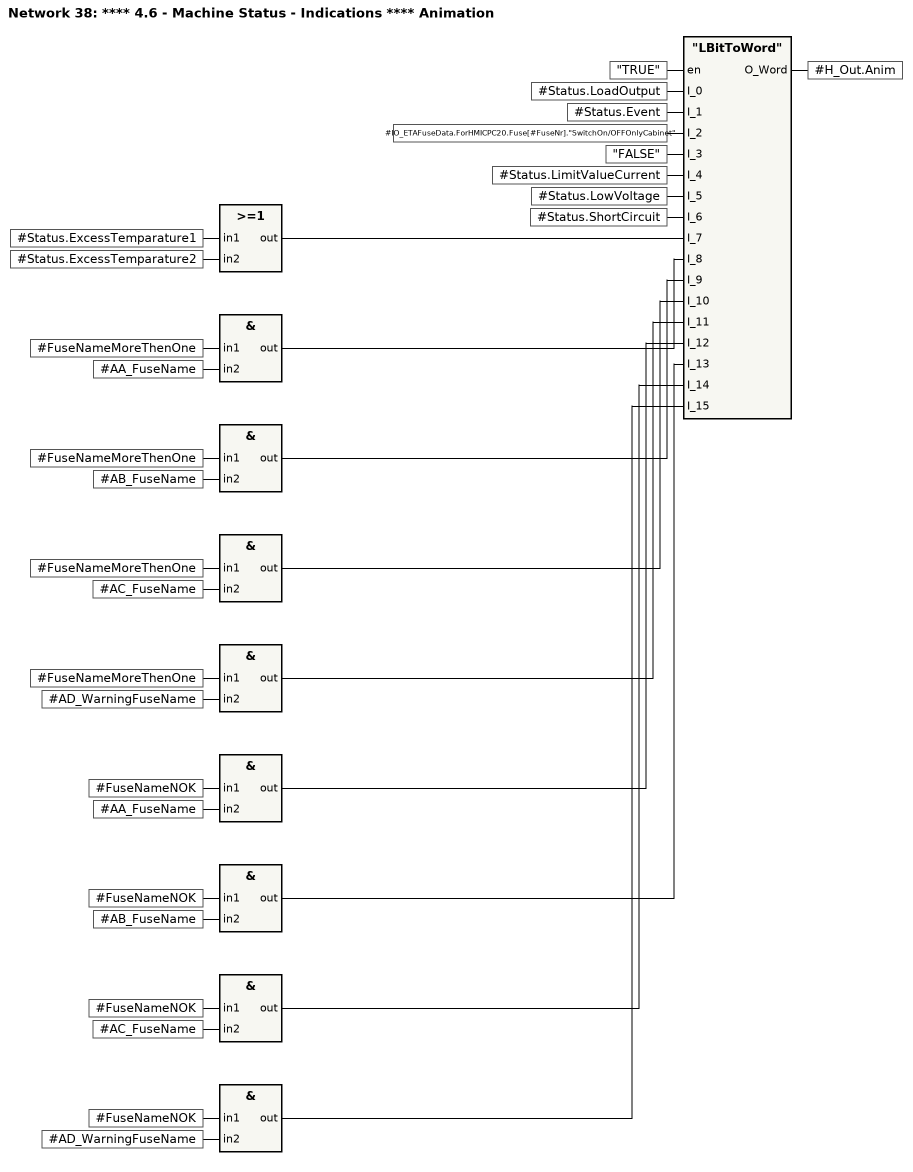
   IF "TRUE" THEN
       "LBitToWord"(I_0 := #Status.LoadOutput,
                    I_1 := #Status.Event,
                    I_2 := #IO_ETAFuseData.ForHMICPC20.Fuse[#FuseNr]."SwitchOn/OFFOnlyCabinet",
                    I_3 := "FALSE",
                    I_4 := #Status.LimitValueCurrent,
                    I_5 := #Status.LowVoltage,
                    I_6 := #Status.ShortCircuit,
                    I_7 := #Status.ExcessTemparature1 OR #Status.ExcessTemparature2,
                    I_8 := #FuseNameMoreThenOne AND #AA_FuseName,
                    I_9 := #FuseNameMoreThenOne AND #AB_FuseName,
                    I_10 := #FuseNameMoreThenOne AND #AC_FuseName,
                    I_11 := #FuseNameMoreThenOne AND #AD_WarningFuseName,
                    I_12 := #FuseNameNOK AND #AA_FuseName,
                    I_13 := #FuseNameNOK AND #AB_FuseName,
                    I_14 := #FuseNameNOK AND #AC_FuseName,
                    I_15 := #FuseNameNOK AND #AD_WarningFuseName,
                    O_Word => #H_Out.Anim);
   END_IF;
END_REGION

REGION Network 39: **** 4.6 - Machine Status - Indications **** Animation2
   // Animation
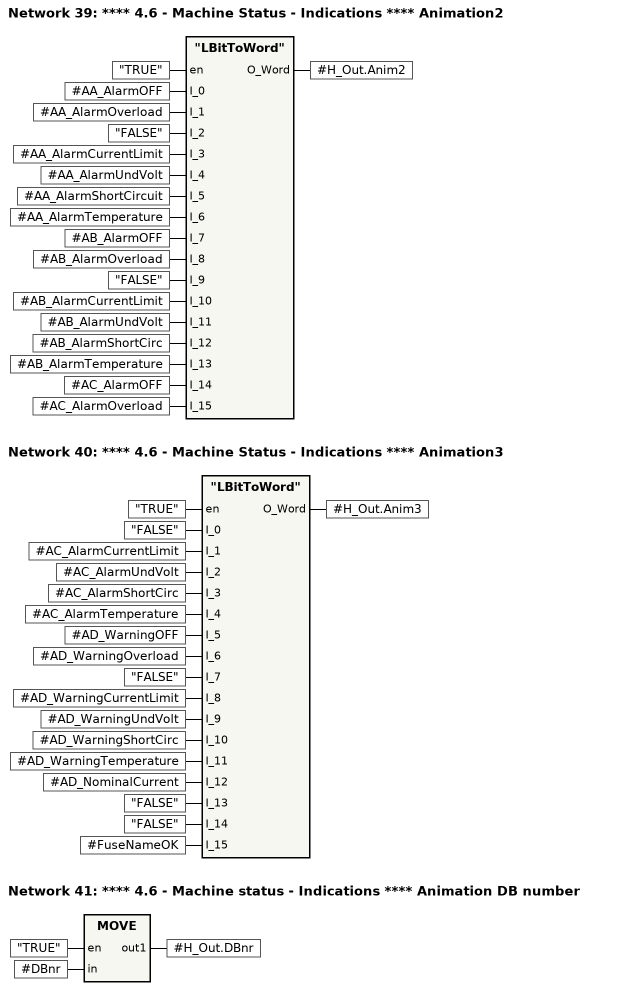
   IF "TRUE" THEN
       "LBitToWord"(I_0 := #AA_AlarmOFF,
                    I_1 := #AA_AlarmOverload,
                    I_2 := "FALSE",
                    I_3 := #AA_AlarmCurrentLimit,
                    I_4 := #AA_AlarmUndVolt,
                    I_5 := #AA_AlarmShortCircuit,
                    I_6 := #AA_AlarmTemperature,
                    I_7 := #AB_AlarmOFF,
                    I_8 := #AB_AlarmOverload,
                    I_9 := "FALSE",
                    I_10 := #AB_AlarmCurrentLimit,
                    I_11 := #AB_AlarmUndVolt,
                    I_12 := #AB_AlarmShortCirc,
                    I_13 := #AB_AlarmTemperature,
                    I_14 := #AC_AlarmOFF,
                    I_15 := #AC_AlarmOverload,
                    O_Word => #H_Out.Anim2);
   END_IF;
END_REGION

REGION Network 40: **** 4.6 - Machine Status - Indications **** Animation3
   // Animation
   IF "TRUE" THEN
       "LBitToWord"(I_0 := "FALSE",
                    I_1 := #AC_AlarmCurrentLimit,
                    I_2 := #AC_AlarmUndVolt,
                    I_3 := #AC_AlarmShortCirc,
                    I_4 := #AC_AlarmTemperature,
                    I_5 := #AD_WarningOFF,
                    I_6 := #AD_WarningOverload,
                    I_7 := "FALSE",
                    I_8 := #AD_WarningCurrentLimit,
                    I_9 := #AD_WarningUndVolt,
                    I_10 := #AD_WarningShortCirc,
                    I_11 := #AD_WarningTemperature,
                    I_12 := #AD_NominalCurrent,
                    I_13 := "FALSE",
                    I_14 := "FALSE",
                    I_15 := #FuseNameOK,
                    O_Word => #H_Out.Anim3);
   END_IF;
END_REGION

REGION Network 41: **** 4.6 - Machine status - Indications **** Animation DB number
   // DB number
   IF "TRUE" THEN #H_Out.DBnr := #DBnr; END_IF;
END_REGION

REGION Network 42: **** 4.6 - Machine Status - Indications **** Animation Fuse Info -> Fuse Number = 0
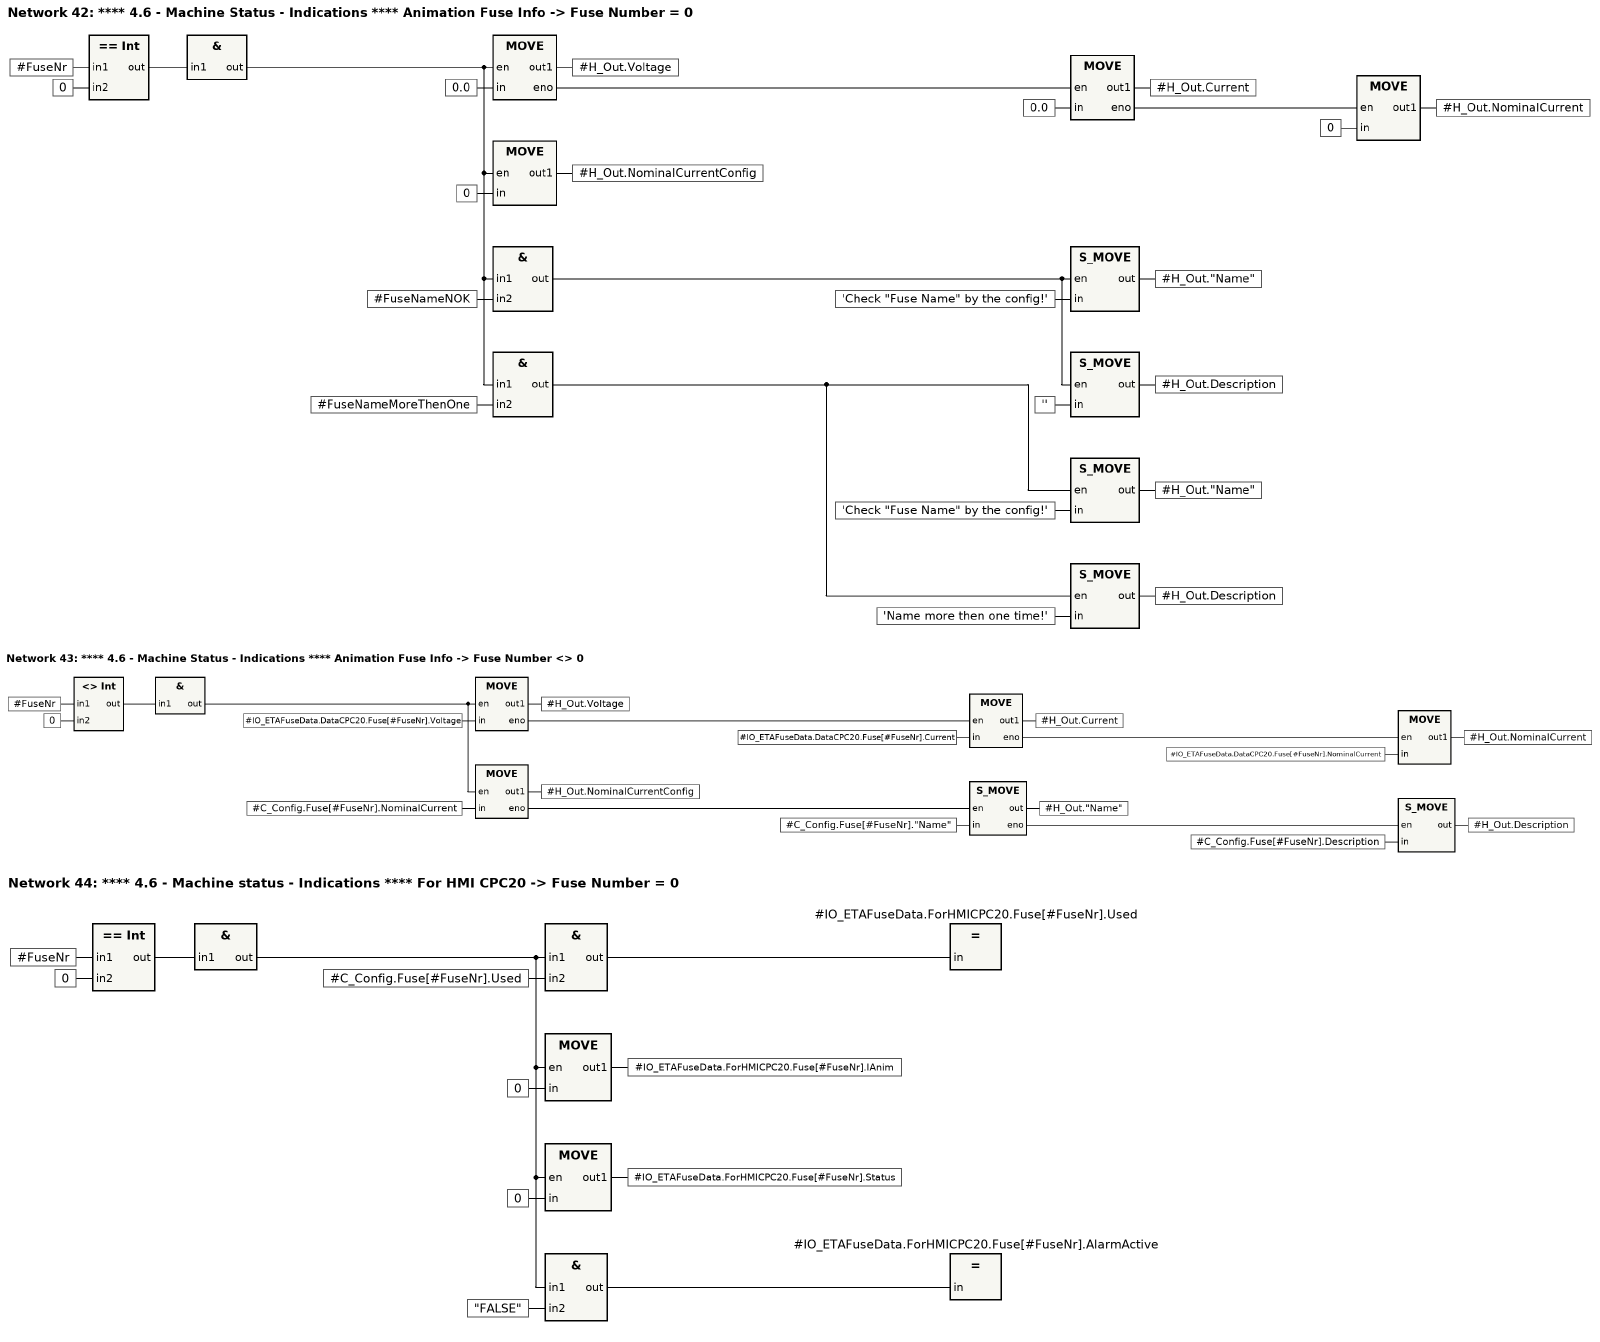
   #_w1 := #FuseNr = 0;
   IF #_w1 THEN
       #H_Out.Voltage := 0.0;
       #H_Out.Current := 0.0;
       #H_Out.NominalCurrent := 0;
       #H_Out.NominalCurrentConfig := 0;
   END_IF;
   IF #_w1 AND #FuseNameNOK THEN
       #H_Out."Name" := 'Check "Fuse Name" by the config!';
       #H_Out.Description := '';
   END_IF;
   IF #_w1 AND #FuseNameMoreThenOne THEN
       #H_Out."Name" := 'Check "Fuse Name" by the config!';
       #H_Out.Description := 'Name more then one time!';
   END_IF;
END_REGION

REGION Network 43: **** 4.6 - Machine Status - Indications **** Animation Fuse Info -> Fuse Number <> 0
   IF #FuseNr <> 0 THEN
       #H_Out.Voltage := #IO_ETAFuseData.DataCPC20.Fuse[#FuseNr].Voltage;
       #H_Out.Current := #IO_ETAFuseData.DataCPC20.Fuse[#FuseNr].Current;
       #H_Out.NominalCurrent := #IO_ETAFuseData.DataCPC20.Fuse[#FuseNr].NominalCurrent;
       #H_Out.NominalCurrentConfig := #C_Config.Fuse[#FuseNr].NominalCurrent;
       #H_Out."Name" := #C_Config.Fuse[#FuseNr]."Name";
       #H_Out.Description := #C_Config.Fuse[#FuseNr].Description;
   END_IF;
END_REGION

REGION Network 44: **** 4.6 - Machine status - Indications **** For HMI CPC20 -> Fuse Number = 0
   #_w1 := #FuseNr = 0;
   #IO_ETAFuseData.ForHMICPC20.Fuse[#FuseNr].Used := #_w1 AND #C_Config.Fuse[#FuseNr].Used;
   IF #_w1 THEN
       #IO_ETAFuseData.ForHMICPC20.Fuse[#FuseNr].IAnim := 0;
       #IO_ETAFuseData.ForHMICPC20.Fuse[#FuseNr].Status := 0;
   END_IF;
   #IO_ETAFuseData.ForHMICPC20.Fuse[#FuseNr].AlarmActive := #_w1 AND "FALSE";
END_REGION

REGION Network 45: **** 4.6 - Machine status - Indications **** For HMI CPC20 -> Fuse Number <> 0
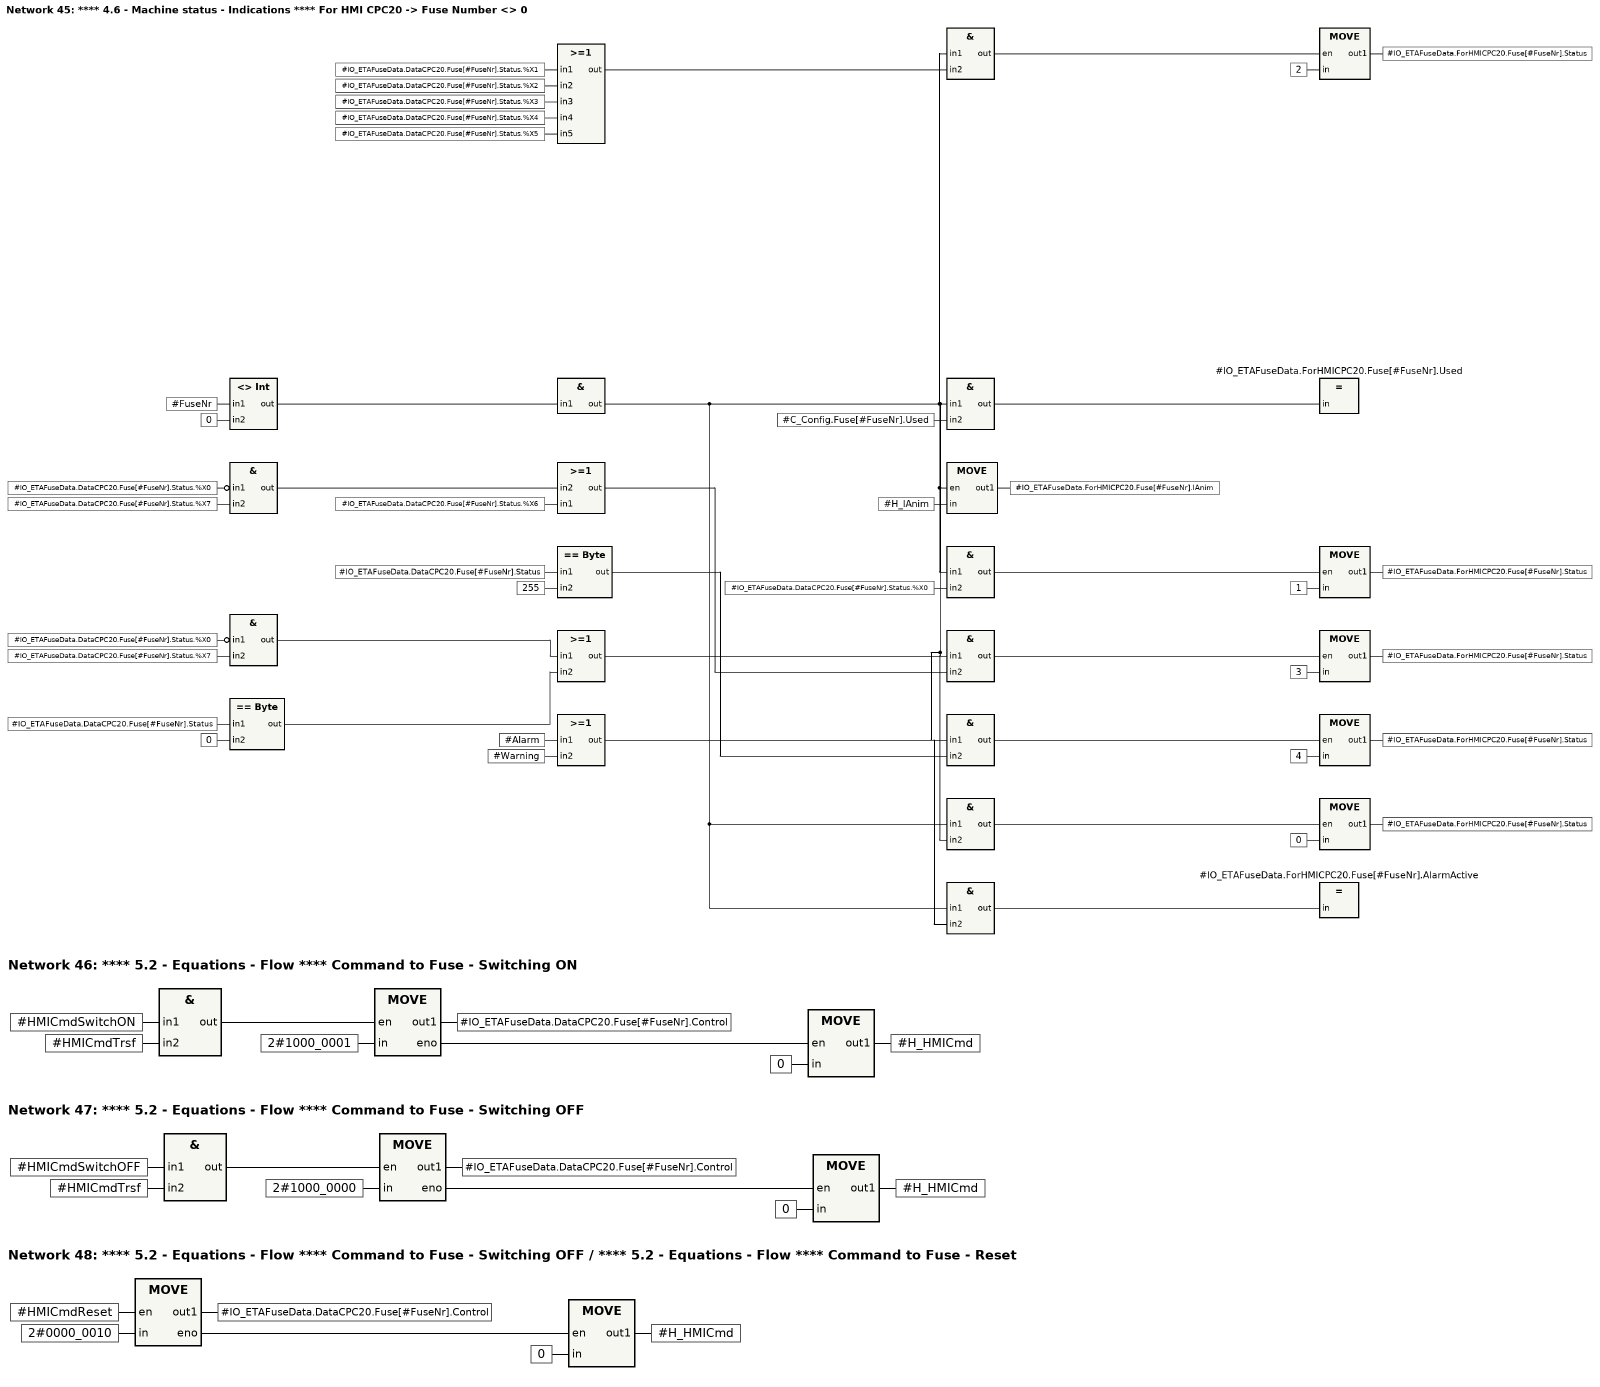
   #_w1 := #FuseNr <> 0;
   #IO_ETAFuseData.ForHMICPC20.Fuse[#FuseNr].Used := #_w1 AND #C_Config.Fuse[#FuseNr].Used;
   IF #_w1 THEN #IO_ETAFuseData.ForHMICPC20.Fuse[#FuseNr].IAnim := #H_IAnim; END_IF;
   IF #_w1 AND #IO_ETAFuseData.DataCPC20.Fuse[#FuseNr].Status.%X0 THEN
       #IO_ETAFuseData.ForHMICPC20.Fuse[#FuseNr].Status := 1;
   END_IF;
   IF #_w1 AND (#IO_ETAFuseData.DataCPC20.Fuse[#FuseNr].Status.%X1 OR #IO_ETAFuseData.DataCPC20.Fuse[#FuseNr].Status.%X2 OR #IO_ETAFuseData.DataCPC20.Fuse[#FuseNr].Status.%X3 OR #IO_ETAFuseData.DataCPC20.Fuse[#FuseNr].Status.%X4 OR #IO_ETAFuseData.DataCPC20.Fuse[#FuseNr].Status.%X5) THEN
       #IO_ETAFuseData.ForHMICPC20.Fuse[#FuseNr].Status := 2;
   END_IF;
   IF #_w1 AND ((NOT #IO_ETAFuseData.DataCPC20.Fuse[#FuseNr].Status.%X0 AND #IO_ETAFuseData.DataCPC20.Fuse[#FuseNr].Status.%X7) OR #IO_ETAFuseData.DataCPC20.Fuse[#FuseNr].Status.%X6) THEN
       #IO_ETAFuseData.ForHMICPC20.Fuse[#FuseNr].Status := 3;
   END_IF;
   IF #_w1 AND (#IO_ETAFuseData.DataCPC20.Fuse[#FuseNr].Status = 255) THEN
       #IO_ETAFuseData.ForHMICPC20.Fuse[#FuseNr].Status := 4;
   END_IF;
   IF #_w1 AND ((NOT #IO_ETAFuseData.DataCPC20.Fuse[#FuseNr].Status.%X0 AND #IO_ETAFuseData.DataCPC20.Fuse[#FuseNr].Status.%X7) OR (#IO_ETAFuseData.DataCPC20.Fuse[#FuseNr].Status = 0)) THEN
       #IO_ETAFuseData.ForHMICPC20.Fuse[#FuseNr].Status := 0;
   END_IF;
   #IO_ETAFuseData.ForHMICPC20.Fuse[#FuseNr].AlarmActive := #_w1 AND (#Alarm OR #Warning);
END_REGION

REGION Network 46: **** 5.2 - Equations - Flow **** Command to Fuse - Switching ON
   // Switching ON
   // ENO of a box is taken as its EN; it also drops when the box reports an error
   IF #HMICmdSwitchON AND #HMICmdTrsf THEN
       #IO_ETAFuseData.DataCPC20.Fuse[#FuseNr].Control := 2#1000_0001;
       #H_HMICmd := 0;
   END_IF;
END_REGION

REGION Network 47: **** 5.2 - Equations - Flow **** Command to Fuse - Switching OFF
   // Switching OFF
   // ENO of a box is taken as its EN; it also drops when the box reports an error
   IF #HMICmdSwitchOFF AND #HMICmdTrsf THEN
       #IO_ETAFuseData.DataCPC20.Fuse[#FuseNr].Control := 2#1000_0000;
       #H_HMICmd := 0;
   END_IF;
END_REGION

REGION Network 48: **** 5.2 - Equations - Flow **** Command to Fuse - Switching OFF / **** 5.2 - Equations - Flow **** Command to Fuse - Reset
   // Switching OFF / Reset
   // ENO of a box is taken as its EN; it also drops when the box reports an error
   IF #HMICmdReset THEN
       #IO_ETAFuseData.DataCPC20.Fuse[#FuseNr].Control := 2#0000_0010;
       #H_HMICmd := 0;
   END_IF;
END_REGION

REGION Network 49: **** 5.2 - Equations - Flow **** Command to Fuse - Reset Control
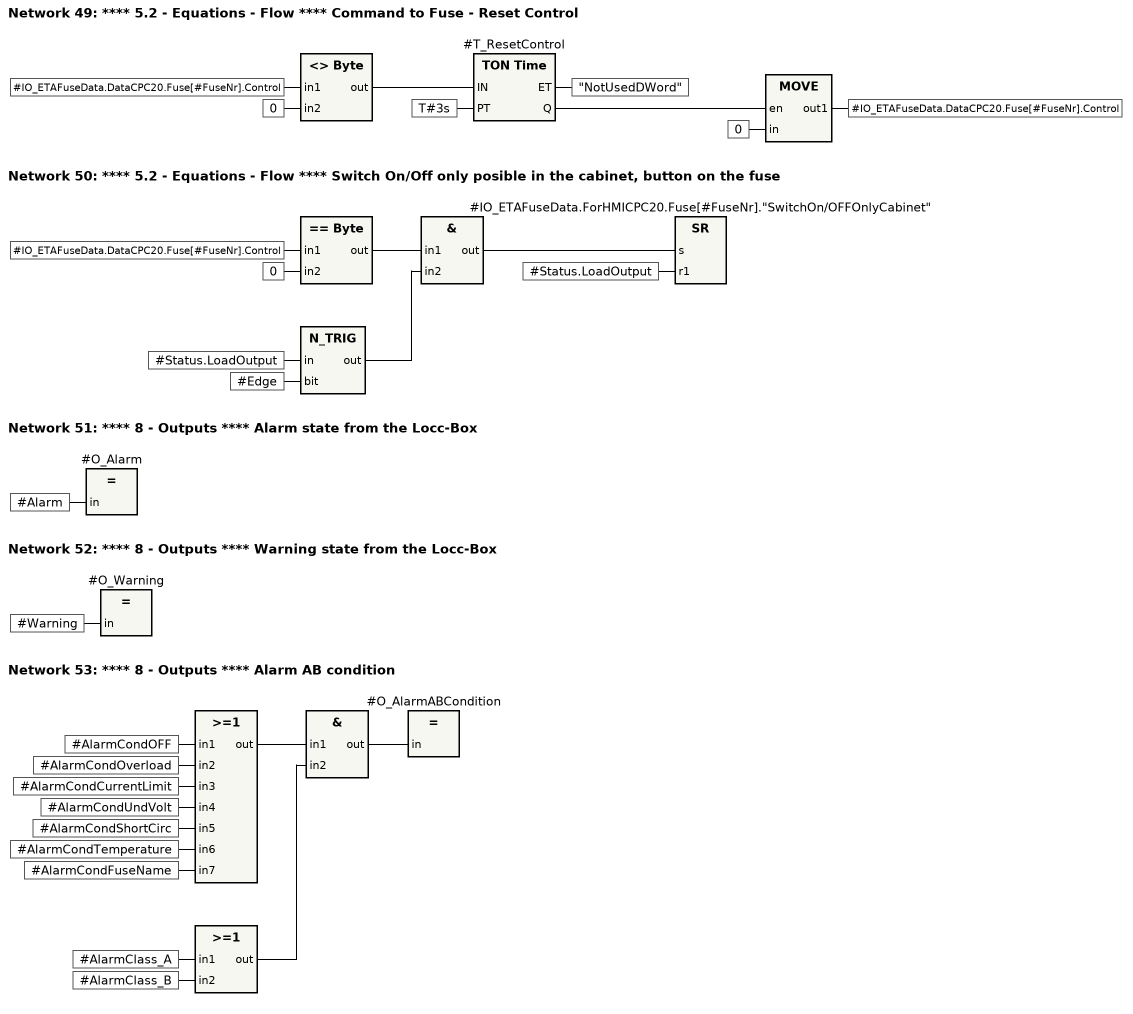
   #T_ResetControl(IN := #IO_ETAFuseData.DataCPC20.Fuse[#FuseNr].Control <> 0, PT := T#3s, ET => "NotUsedDWord");   // TON
   IF #T_ResetControl.Q THEN #IO_ETAFuseData.DataCPC20.Fuse[#FuseNr].Control := 0; END_IF;
END_REGION

REGION Network 50: **** 5.2 - Equations - Flow **** Switch On/Off only posible in the cabinet, button on the fuse
   #_w1 := NOT #Status.LoadOutput AND #Edge;   // falling edge
   #Edge := #Status.LoadOutput;
   IF (#IO_ETAFuseData.DataCPC20.Fuse[#FuseNr].Control = 0) AND #_w1 THEN
       #IO_ETAFuseData.ForHMICPC20.Fuse[#FuseNr]."SwitchOn/OFFOnlyCabinet" := TRUE;   // SR flip-flop
   END_IF;
   IF #Status.LoadOutput THEN
       #IO_ETAFuseData.ForHMICPC20.Fuse[#FuseNr]."SwitchOn/OFFOnlyCabinet" := FALSE;
   END_IF;
END_REGION

REGION Network 51: **** 8 - Outputs **** Alarm state from the Locc-Box
   // Alarm state from the Locc-Box
   #O_Alarm := #Alarm;
END_REGION

REGION Network 52: **** 8 - Outputs **** Warning state from the Locc-Box
   // Warning state from the Locc-Box
   #O_Warning := #Warning;
END_REGION

REGION Network 53: **** 8 - Outputs **** Alarm AB condition
   // Alarm AB condition
   #O_AlarmABCondition := (#AlarmCondOFF OR #AlarmCondOverload OR #AlarmCondCurrentLimit OR #AlarmCondUndVolt OR #AlarmCondShortCirc OR #AlarmCondTemperature OR #AlarmCondFuseName) AND (#AlarmClass_A OR #AlarmClass_B);
END_REGION

REGION Network 54: **** 9.2 - Alarm DWord**** Alarm To DWord
   // Alarm Word
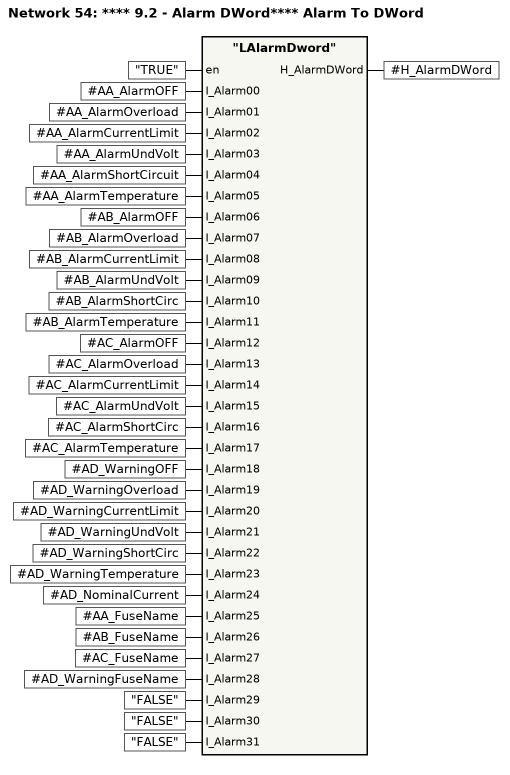
   IF "TRUE" THEN
       "LAlarmDword"(I_Alarm00 := #AA_AlarmOFF,
                     I_Alarm01 := #AA_AlarmOverload,
                     I_Alarm02 := #AA_AlarmCurrentLimit,
                     I_Alarm03 := #AA_AlarmUndVolt,
                     I_Alarm04 := #AA_AlarmShortCircuit,
                     I_Alarm05 := #AA_AlarmTemperature,
                     I_Alarm06 := #AB_AlarmOFF,
                     I_Alarm07 := #AB_AlarmOverload,
                     I_Alarm08 := #AB_AlarmCurrentLimit,
                     I_Alarm09 := #AB_AlarmUndVolt,
                     I_Alarm10 := #AB_AlarmShortCirc,
                     I_Alarm11 := #AB_AlarmTemperature,
                     I_Alarm12 := #AC_AlarmOFF,
                     I_Alarm13 := #AC_AlarmOverload,
                     I_Alarm14 := #AC_AlarmCurrentLimit,
                     I_Alarm15 := #AC_AlarmUndVolt,
                     I_Alarm16 := #AC_AlarmShortCirc,
                     I_Alarm17 := #AC_AlarmTemperature,
                     I_Alarm18 := #AD_WarningOFF,
                     I_Alarm19 := #AD_WarningOverload,
                     I_Alarm20 := #AD_WarningCurrentLimit,
                     I_Alarm21 := #AD_WarningUndVolt,
                     I_Alarm22 := #AD_WarningShortCirc,
                     I_Alarm23 := #AD_WarningTemperature,
                     I_Alarm24 := #AD_NominalCurrent,
                     I_Alarm25 := #AA_FuseName,
                     I_Alarm26 := #AB_FuseName,
                     I_Alarm27 := #AC_FuseName,
                     I_Alarm28 := #AD_WarningFuseName,
                     I_Alarm29 := "FALSE",
                     I_Alarm30 := "FALSE",
                     I_Alarm31 := "FALSE",
                     H_AlarmDWord => #H_AlarmDWord);
   END_IF;
END_REGION
END_FUNCTION_BLOCK

FUNCTION_BLOCK "LGapControlAlarm"   // FB1415, FBD
TITLE = LGapControlAlarm
{ S7_Optimized_Access := 'FALSE' }
AUTHOR : VCC
FAMILY : AlarmHnd
NAME : GapCtrl
VERSION : 1.0
// ================================================================================
// This module is used everywhere one alarm shall be generated when one input 
// photocell becomes false and this photocell signal has to be checked during 
// transfer.
// If the alarm is enable, the photocell may not be deactivated by means of 
// breaking the ray.
// This FB also check the consistency of the photocell. During the period we are 
// sure the photocell must be activated (transfer), the input of the photocell is 
// checked on activity.
// Alarm is disable from HMI, a boolean output is available to inform the upper 
// level and do action in the Alarm summary.
// When the conditions to generate the alarm is disappear, a boolean output is 
// available to inform the upper level that the alarm can be reset.
// The alarm is reset by means of the AlarmResetPB signal.
// ================================================================================
// stored: AutoNumber false, IsIECCheckEnabled false, SetENOAutomatically False, UDAEnableTagReadback false
   VAR_INPUT
      I_GapControl { ExternalAccessible := 'False'; ExternalVisible := 'False'; ExternalWritable := 'False'} : Bool;   // Input signal of the alarm
      I_CheckGapCtrlTrueCond { ExternalAccessible := 'False'; ExternalVisible := 'False'; ExternalWritable := 'False'} : Bool;   // Condition to check gap control photocell on TRUE
      I_CheckGapCtrlFalseCond { ExternalAccessible := 'False'; ExternalVisible := 'False'; ExternalWritable := 'False'} : Bool;   // Condition ot check gap control photocell on FALSE
      I_EnableAlarm { ExternalAccessible := 'False'; ExternalVisible := 'False'; ExternalWritable := 'False'} : Bool := TRUE;   // Enable alarm from upper level
      I_Invisible { ExternalAccessible := 'False'; ExternalVisible := 'False'; ExternalWritable := 'False'} : Bool;   // Invisible
      I_AlarmResetPB { ExternalAccessible := 'False'; ExternalVisible := 'False'; ExternalWritable := 'False'} : Bool;   // Alarm reset pushbutton is activated
   END_VAR
   VAR_OUTPUT
      O_GapControlAlm { ExternalAccessible := 'False'; ExternalVisible := 'False'; ExternalWritable := 'False'} : Bool;   // Gap control Alarm
      O_GapControlTrueAlm { ExternalAccessible := 'False'; ExternalVisible := 'False'; ExternalWritable := 'False'} : Bool;   // Gap control True Alarm
      O_GapControlFalseAlm { ExternalAccessible := 'False'; ExternalVisible := 'False'; ExternalWritable := 'False'} : Bool;   // Gap control False Alarm
      O_AlarmDisabled { ExternalAccessible := 'False'; ExternalVisible := 'False'; ExternalWritable := 'False'} : Bool;   // Alarm disabled from HMI
      O_AlarmABCondition { ExternalAccessible := 'False'; ExternalVisible := 'False'; ExternalWritable := 'False'} : Bool;   // Alarm AB condition
      H_IAnim { ExternalAccessible := 'False'; ExternalVisible := 'False'; ExternalWritable := 'False'} : Word;
   END_VAR
   VAR DB_SPECIFIC
      H_In : Struct   // HMI
         DisableAlarm : Bool;   // Disable alarm from HMI
      END_STRUCT;
      H_Out : Struct   // HMI
         Anim : Word;   // HMI Animation of the object
      END_STRUCT;
      GapControlAlm { ExternalAccessible := 'False'; ExternalVisible := 'False'; ExternalWritable := 'False'} : Bool;   // Gap control Alarm
      GapControlAlmCond { ExternalAccessible := 'False'; ExternalVisible := 'False'; ExternalWritable := 'False'} : Bool;   // Gap control Alarm condition
      PCheckGapTrue { ExternalAccessible := 'False'; ExternalVisible := 'False'; ExternalWritable := 'False'} : Bool;   // Pulse Check detection on True signal
      GapControlTrueMem { ExternalAccessible := 'False'; ExternalVisible := 'False'; ExternalWritable := 'False'} : Bool;   // Memory Gap control on True signal
      GapControlTrueAlm { ExternalAccessible := 'False'; ExternalVisible := 'False'; ExternalWritable := 'False'} : Bool;   // Gap control alarm on True
      GapControlTrueAlmCond { ExternalAccessible := 'False'; ExternalVisible := 'False'; ExternalWritable := 'False'} : Bool;   // Alarm condition of Gap Control True Alarm
      PCheckGapfalse { ExternalAccessible := 'False'; ExternalVisible := 'False'; ExternalWritable := 'False'} : Bool;   // Pulse Check detection on False signal
      GapControlFalseMem { ExternalAccessible := 'False'; ExternalVisible := 'False'; ExternalWritable := 'False'} : Bool;   // Memory Gap control on False signal
      GapControlFalseAlm { ExternalAccessible := 'False'; ExternalVisible := 'False'; ExternalWritable := 'False'} : Bool;   // Gap control alarm on False
      GapControlFalseAlmCond { ExternalAccessible := 'False'; ExternalVisible := 'False'; ExternalWritable := 'False'} : Bool;   // Alarm condition of Gap Control False Alarm
   END_VAR
   VAR_TEMP   // added for the SCL form of the ladder/FBD networks
      _w1 : Bool;
   END_VAR
BEGIN

REGION Network 1: **** 2.2 - Alarms - Alarms Generation **** Condition of the Gap control alarm for the Normal CLOSED input
   // Condition of the Gap control alarm for the Normal CLOSED input
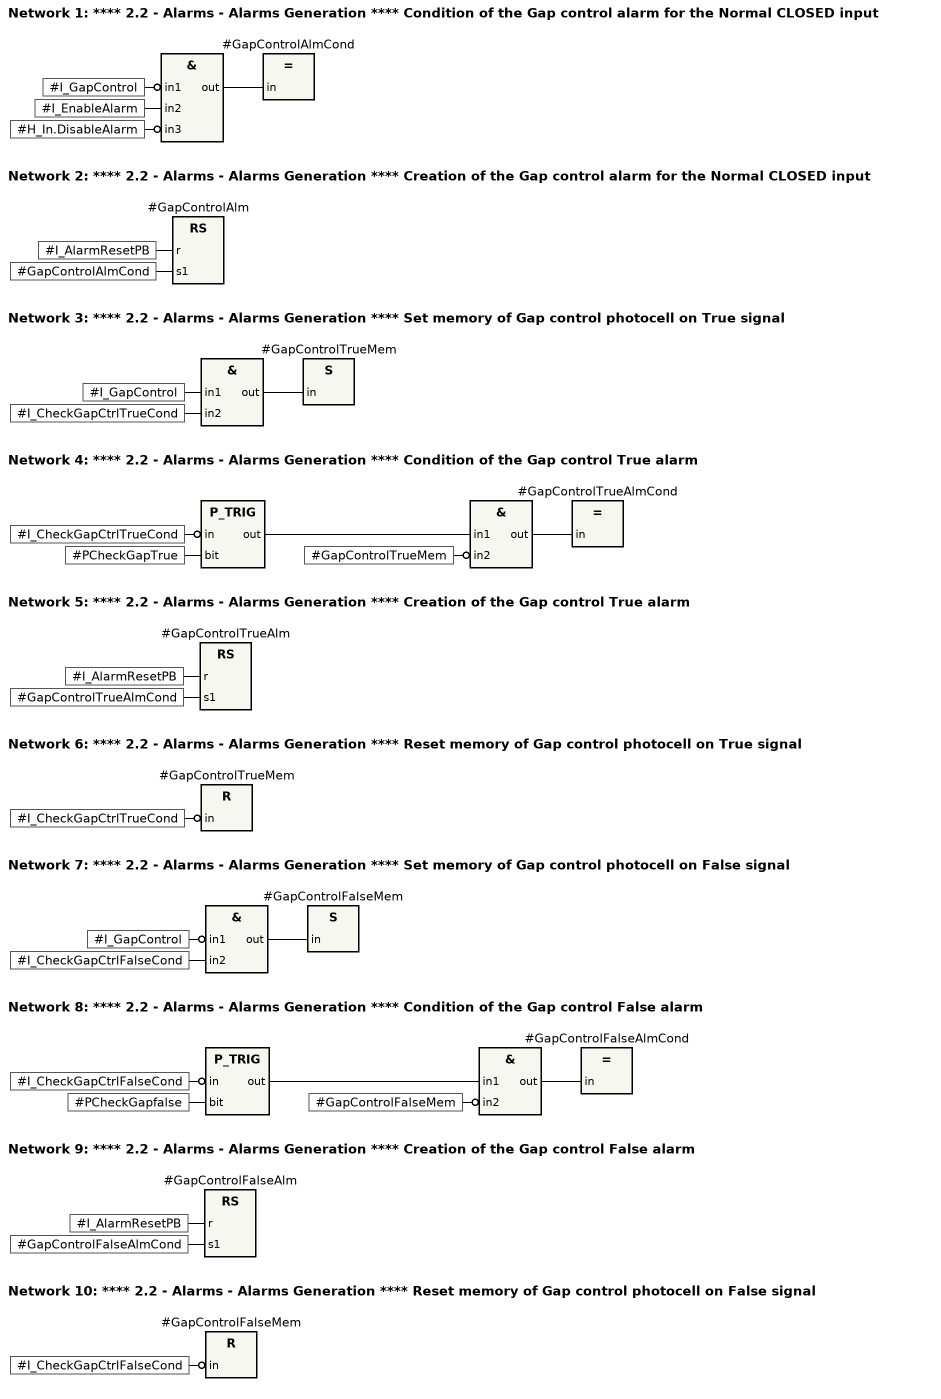
   #GapControlAlmCond := NOT #I_GapControl AND #I_EnableAlarm AND NOT #H_In.DisableAlarm;
END_REGION

REGION Network 2: **** 2.2 - Alarms - Alarms Generation **** Creation of the Gap control alarm for the Normal CLOSED input
   // Creation of the Gap control alarm for the Normal CLOSED input
   IF #I_AlarmResetPB THEN
       #GapControlAlm := FALSE;   // RS flip-flop
   END_IF;
   IF #GapControlAlmCond THEN #GapControlAlm := TRUE; END_IF;
END_REGION

REGION Network 3: **** 2.2 - Alarms - Alarms Generation **** Set memory of Gap control photocell on True signal
   // Set memory of Gap control photocell on True signal
   IF #I_GapControl AND #I_CheckGapCtrlTrueCond THEN #GapControlTrueMem := TRUE; END_IF;
END_REGION

REGION Network 4: **** 2.2 - Alarms - Alarms Generation **** Condition of the Gap control True alarm
   // Condition of the Gap control True alarm
   #_w1 := NOT #I_CheckGapCtrlTrueCond AND NOT #PCheckGapTrue;   // rising edge
   #PCheckGapTrue := NOT #I_CheckGapCtrlTrueCond;
   #GapControlTrueAlmCond := #_w1 AND NOT #GapControlTrueMem;
END_REGION

REGION Network 5: **** 2.2 - Alarms - Alarms Generation **** Creation of the Gap control True alarm
   // Creation of the Gap control True alarm
   IF #I_AlarmResetPB THEN
       #GapControlTrueAlm := FALSE;   // RS flip-flop
   END_IF;
   IF #GapControlTrueAlmCond THEN #GapControlTrueAlm := TRUE; END_IF;
END_REGION

REGION Network 6: **** 2.2 - Alarms - Alarms Generation **** Reset memory of Gap control photocell on True signal
   // Reset memory of Gap control photocell on True signal
   IF NOT #I_CheckGapCtrlTrueCond THEN #GapControlTrueMem := FALSE; END_IF;
END_REGION

REGION Network 7: **** 2.2 - Alarms - Alarms Generation **** Set memory of Gap control photocell on False signal
   // Set memory of Gap control photocell on False signal
   IF NOT #I_GapControl AND #I_CheckGapCtrlFalseCond THEN #GapControlFalseMem := TRUE; END_IF;
END_REGION

REGION Network 8: **** 2.2 - Alarms - Alarms Generation **** Condition of the Gap control False alarm
   // Condition of the Gap control False alarm
   #_w1 := NOT #I_CheckGapCtrlFalseCond AND NOT #PCheckGapfalse;   // rising edge
   #PCheckGapfalse := NOT #I_CheckGapCtrlFalseCond;
   #GapControlFalseAlmCond := #_w1 AND NOT #GapControlFalseMem;
END_REGION

REGION Network 9: **** 2.2 - Alarms - Alarms Generation **** Creation of the Gap control False alarm
   // Creation of the Gap control False alarm
   IF #I_AlarmResetPB THEN
       #GapControlFalseAlm := FALSE;   // RS flip-flop
   END_IF;
   IF #GapControlFalseAlmCond THEN #GapControlFalseAlm := TRUE; END_IF;
END_REGION

REGION Network 10: **** 2.2 - Alarms - Alarms Generation **** Reset memory of Gap control photocell on False signal
   // Reset memory of Gap control photocell on False signal
   IF NOT #I_CheckGapCtrlFalseCond THEN #GapControlFalseMem := FALSE; END_IF;
END_REGION

REGION Network 11: **** 4.6 - Mashine Status - Indications **** Icon Animation
   // Icon Animation
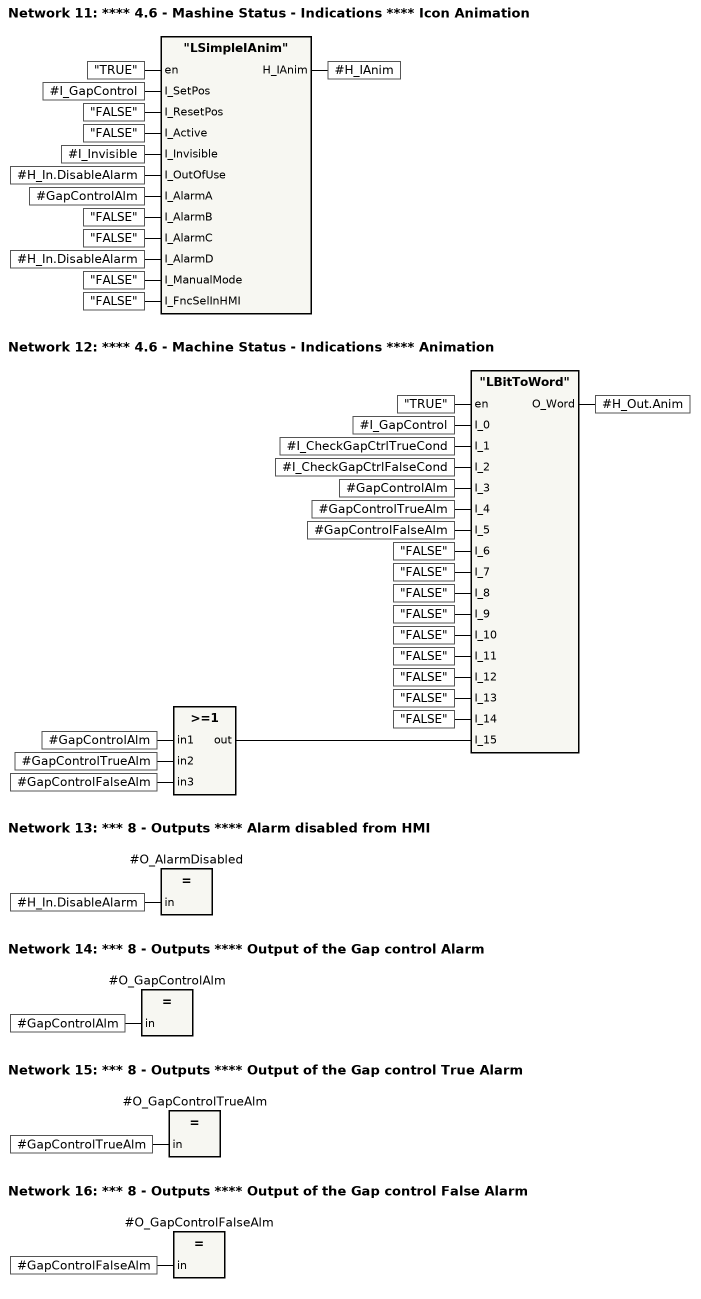
   IF "TRUE" THEN
       "LSimpleIAnim"(I_SetPos := #I_GapControl,
                      I_ResetPos := "FALSE",
                      I_Active := "FALSE",
                      I_Invisible := #I_Invisible,
                      I_OutOfUse := #H_In.DisableAlarm,
                      I_AlarmA := #GapControlAlm,
                      I_AlarmB := "FALSE",
                      I_AlarmC := "FALSE",
                      I_AlarmD := #H_In.DisableAlarm,
                      I_ManualMode := "FALSE",
                      I_FncSelInHMI := "FALSE",
                      H_IAnim => #H_IAnim);
   END_IF;
END_REGION

REGION Network 12: **** 4.6 - Machine Status - Indications **** Animation
   // Animation
   IF "TRUE" THEN
       "LBitToWord"(I_0 := #I_GapControl,
                    I_1 := #I_CheckGapCtrlTrueCond,
                    I_2 := #I_CheckGapCtrlFalseCond,
                    I_3 := #GapControlAlm,
                    I_4 := #GapControlTrueAlm,
                    I_5 := #GapControlFalseAlm,
                    I_6 := "FALSE",
                    I_7 := "FALSE",
                    I_8 := "FALSE",
                    I_9 := "FALSE",
                    I_10 := "FALSE",
                    I_11 := "FALSE",
                    I_12 := "FALSE",
                    I_13 := "FALSE",
                    I_14 := "FALSE",
                    I_15 := #GapControlAlm OR #GapControlTrueAlm OR #GapControlFalseAlm,
                    O_Word => #H_Out.Anim);
   END_IF;
END_REGION

REGION Network 13: *** 8 - Outputs **** Alarm disabled from HMI
   // Alarm disabled from HMI
   #O_AlarmDisabled := #H_In.DisableAlarm;
END_REGION

REGION Network 14: *** 8 - Outputs **** Output of the Gap control Alarm
   // Output of the Gap control Alarm
   #O_GapControlAlm := #GapControlAlm;
END_REGION

REGION Network 15: *** 8 - Outputs **** Output of the Gap control True Alarm
   // Output of the Gap control True Alarm
   #O_GapControlTrueAlm := #GapControlTrueAlm;
END_REGION

REGION Network 16: *** 8 - Outputs **** Output of the Gap control False Alarm
   // Output of the Gap control False Alarm
   #O_GapControlFalseAlm := #GapControlFalseAlm;
END_REGION

REGION Network 17: **** 8 - Outputs **** Alarm resetable
   // Alarm resetable
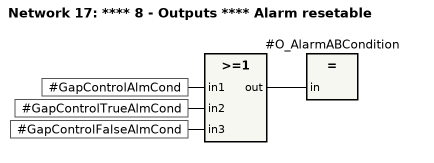
   #O_AlarmABCondition := #GapControlAlmCond OR #GapControlTrueAlmCond OR #GapControlFalseAlmCond;
END_REGION
END_FUNCTION_BLOCK

FUNCTION_BLOCK "LAcofDet"   // FB1416, FBD
TITLE = LAcofDet
{ S7_Optimized_Access := 'FALSE' }
AUTHOR : VCC
FAMILY : Actuator
NAME : LAcofDet
VERSION : 1.0
// ===============================================================================
// This module handles a partdetection with all his functions and alarms
// Functions are DetCheckOn, DetCheckOff and EnableAlarm
// Outputs are DetAlarm and DetSim signal
// ===============================================================================
// stored: AutoNumber false, IsIECCheckEnabled false, SetENOAutomatically False, UDAEnableTagReadback false
   VAR_INPUT
      I_Input { ExternalAccessible := 'False'; ExternalVisible := 'False'; ExternalWritable := 'False'} : Bool;   // Actual input from sensor
      I_SignalCheckOn { ExternalAccessible := 'False'; ExternalVisible := 'False'; ExternalWritable := 'False'} : Bool;   // Signal to check signal is on
      I_SignalCheckOff { ExternalAccessible := 'False'; ExternalVisible := 'False'; ExternalWritable := 'False'} : Bool;   // Signal to check signal is off
      I_MaxAcofTime { ExternalAccessible := 'False'; ExternalVisible := 'False'; ExternalWritable := 'False'} : DInt;   // Maximum Time (ms) that the function may run (create overtime)
      I_AlarmClass { ExternalAccessible := 'False'; ExternalVisible := 'False'; ExternalWritable := 'False'} : Char;   // Alarm class -> A - B - C - D or E
      I_EnableAlarm { ExternalAccessible := 'False'; ExternalVisible := 'False'; ExternalWritable := 'False'} : Bool;   // Enable alarms
      I_Simulate { ExternalAccessible := 'False'; ExternalVisible := 'False'; ExternalWritable := 'False'} : Bool;   // Simulate modus
      I_AlarmResetPB { ExternalAccessible := 'False'; ExternalVisible := 'False'; ExternalWritable := 'False'} : Bool;   // Alarm reset pushbutton is activated
      I_Invisible { ExternalAccessible := 'False'; ExternalVisible := 'False'; ExternalWritable := 'False'} : Bool;   // Invisible
      C_DisableViaHMI { ExternalAccessible := 'False'; ExternalVisible := 'False'; ExternalWritable := 'False'} : Bool;   // Config to enable/disable the detection via the HMI
   END_VAR
   VAR_OUTPUT
      O_DetOn { ExternalAccessible := 'False'; ExternalVisible := 'False'; ExternalWritable := 'False'} : Bool;   // Detection signal to use in program
      O_Alarm { ExternalAccessible := 'False'; ExternalVisible := 'False'; ExternalWritable := 'False'} : Bool;   // Detection alarm
      O_AlarmABCondition { ExternalAccessible := 'False'; ExternalVisible := 'False'; ExternalWritable := 'False'} : Bool;   // Alarm AB condition
      O_AlarmDisabled { ExternalAccessible := 'False'; ExternalVisible := 'False'; ExternalWritable := 'False'} : Bool;   // Alarm disabled from HMI
      H_IAnim { ExternalAccessible := 'False'; ExternalVisible := 'False'; ExternalWritable := 'False'} : DWord;   // For animation of the icon
   END_VAR
   VAR DB_SPECIFIC
      H_In : Struct   // HMI
         DisableAlarm : Bool;   // Disable alarm from HMI
      END_STRUCT;
      H_Out : Struct   // HMI
         Anim : Word;   // HMI Animation of the object
         DBnr : Int;   // HMI Animation DB number
      END_STRUCT;
      DetOn { ExternalAccessible := 'False'; ExternalVisible := 'False'; ExternalWritable := 'False'} : Bool;   // Static variable of O_DetOn
      DetOvtAlarm { ExternalAccessible := 'False'; ExternalVisible := 'False'; ExternalWritable := 'False'} : Bool;   // Static variable of O_DetAlarm
      Alarm { ExternalAccessible := 'False'; ExternalVisible := 'False'; ExternalWritable := 'False'} : Bool;   // Alarm condition
      AlarmDisabled { ExternalAccessible := 'False'; ExternalVisible := 'False'; ExternalWritable := 'False'} : Bool;   // Alarm disabled from HMI
      AlarmClass_A { ExternalAccessible := 'False'; ExternalVisible := 'False'; ExternalWritable := 'False'} : Bool;   // The alarm is from alarm class A
      AlarmClass_B { ExternalAccessible := 'False'; ExternalVisible := 'False'; ExternalWritable := 'False'} : Bool;   // The alarm is from alarm class B
      AlarmClass_C { ExternalAccessible := 'False'; ExternalVisible := 'False'; ExternalWritable := 'False'} : Bool;   // The alarm is from alarm class C
      AlarmClass_D { ExternalAccessible := 'False'; ExternalVisible := 'False'; ExternalWritable := 'False'} : Bool;   // The alarm is from alarm class D
      AlarmClass_E { ExternalAccessible := 'False'; ExternalVisible := 'False'; ExternalWritable := 'False'} : Bool;   // The alarm is from alarm class E
      DBnr { ExternalAccessible := 'False'; ExternalVisible := 'False'; ExternalWritable := 'False'} : Int;   // HMI DB number
   END_VAR
   VAR
      MaxTimeTimer { ExternalAccessible := 'False'; ExternalVisible := 'False'; ExternalWritable := 'False'; S7_SetPoint := 'True'} : "LTimer";   // Creating alarm overtime
   END_VAR
BEGIN

NETWORK
TITLE = **** 1 - Inputs **** DB number
// DB number
      L     DINO;
      T     #DBnr;

NETWORK
TITLE = **** 1 - Inputs **** Alarm class
// Alarm class
// Alarm class = E
      L     #I_AlarmClass;
      L     'E';
      ==I;
      =     #AlarmClass_E;

// Alarm class = D
      L     #I_AlarmClass;
      L     'D';
      ==I;
      =     #AlarmClass_D;

// Alarm class = C
      L     #I_AlarmClass;
      L     'C';
      ==I;
      =     #AlarmClass_C;

// Alarm class = B
      L     #I_AlarmClass;
      L     'B';
      ==I;
      =     #AlarmClass_B;

// Alarm class = A
      AN    #AlarmClass_B;
      AN    #AlarmClass_C;
      AN    #AlarmClass_D;
      AN    #AlarmClass_E;
      =     #AlarmClass_A;


REGION Network 3: **** 2.2 - Alarms - Alarm generation **** Creating alarm overtime
   // Creating alarm overtime
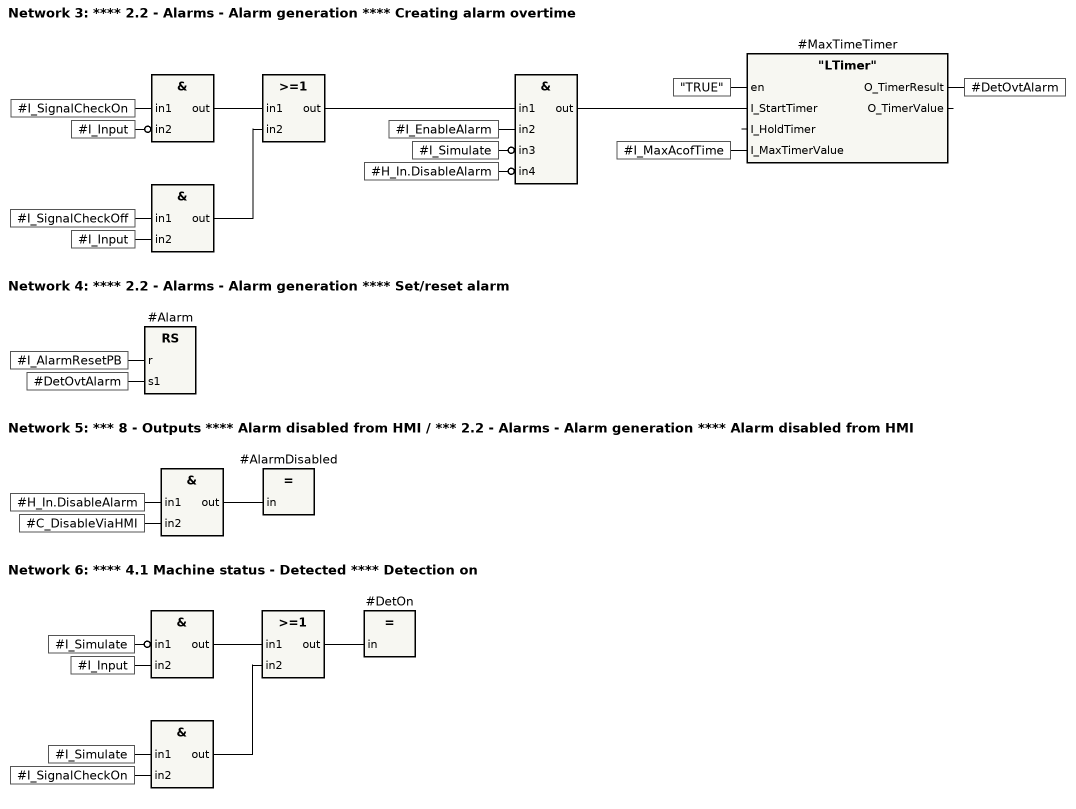
   IF "TRUE" THEN
       #MaxTimeTimer(I_StartTimer := ((#I_SignalCheckOn AND NOT #I_Input) OR (#I_SignalCheckOff AND #I_Input)) AND #I_EnableAlarm AND NOT #I_Simulate AND NOT #H_In.DisableAlarm,   // "LTimer"
                     I_MaxTimerValue := #I_MaxAcofTime,
                     O_TimerResult => #DetOvtAlarm);
   END_IF;
END_REGION

REGION Network 4: **** 2.2 - Alarms - Alarm generation **** Set/reset alarm
   // Set/reset alarm
   IF #I_AlarmResetPB THEN
       #Alarm := FALSE;   // RS flip-flop
   END_IF;
   IF #DetOvtAlarm THEN #Alarm := TRUE; END_IF;
END_REGION

REGION Network 5: *** 8 - Outputs **** Alarm disabled from HMI / *** 2.2 - Alarms - Alarm generation **** Alarm disabled from HMI
   // Alarm disabled from HMI
   #AlarmDisabled := #H_In.DisableAlarm AND #C_DisableViaHMI;
END_REGION

REGION Network 6: **** 4.1 Machine status - Detected **** Detection on
   // Detection on
   #DetOn := (NOT #I_Simulate AND #I_Input) OR (#I_Simulate AND #I_SignalCheckOn);
END_REGION

REGION Network 7: **** 4.6 - Mashine Status - Indications **** Icon Animation
   // Icon Animation
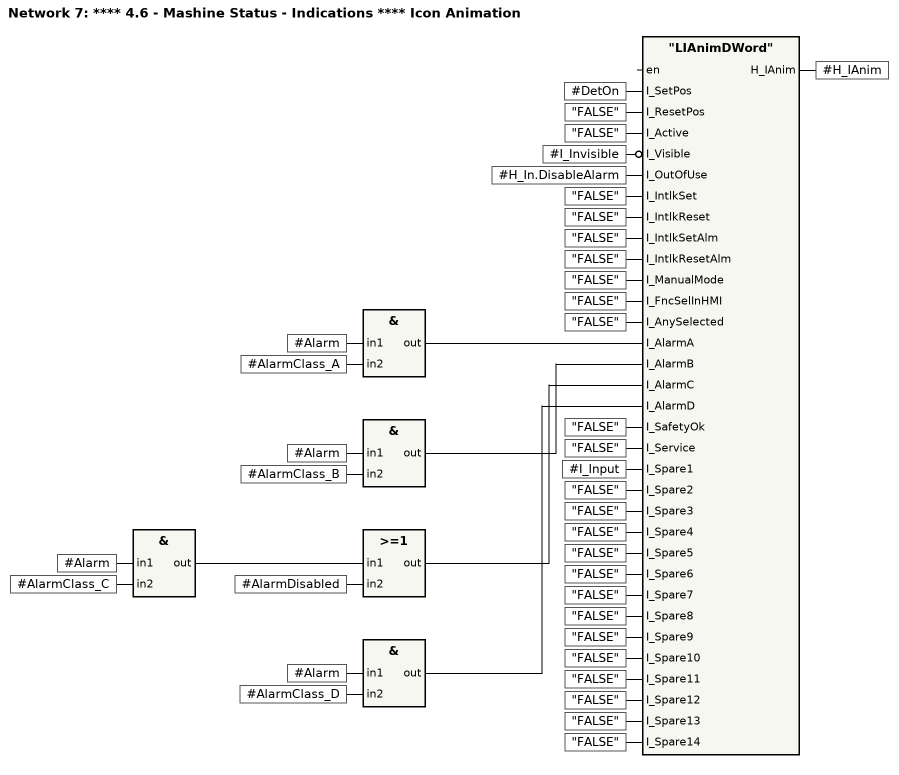
   "LIAnimDWord"(I_SetPos := #DetOn,
                 I_ResetPos := "FALSE",
                 I_Active := "FALSE",
                 I_Visible := NOT #I_Invisible,
                 I_OutOfUse := #H_In.DisableAlarm,
                 I_IntlkSet := "FALSE",
                 I_IntlkReset := "FALSE",
                 I_IntlkSetAlm := "FALSE",
                 I_IntlkResetAlm := "FALSE",
                 I_ManualMode := "FALSE",
                 I_FncSelInHMI := "FALSE",
                 I_AnySelected := "FALSE",
                 I_AlarmA := #Alarm AND #AlarmClass_A,
                 I_AlarmB := #Alarm AND #AlarmClass_B,
                 I_AlarmC := (#Alarm AND #AlarmClass_C) OR #AlarmDisabled,
                 I_AlarmD := #Alarm AND #AlarmClass_D,
                 I_SafetyOk := "FALSE",
                 I_Service := "FALSE",
                 I_Spare1 := #I_Input,
                 I_Spare2 := "FALSE",
                 I_Spare3 := "FALSE",
                 I_Spare4 := "FALSE",
                 I_Spare5 := "FALSE",
                 I_Spare6 := "FALSE",
                 I_Spare7 := "FALSE",
                 I_Spare8 := "FALSE",
                 I_Spare9 := "FALSE",
                 I_Spare10 := "FALSE",
                 I_Spare11 := "FALSE",
                 I_Spare12 := "FALSE",
                 I_Spare13 := "FALSE",
                 I_Spare14 := "FALSE",
                 H_IAnim => #H_IAnim);
END_REGION

REGION Network 8: **** 4.6 - Machine Status - Indications **** Animation
   // Animation
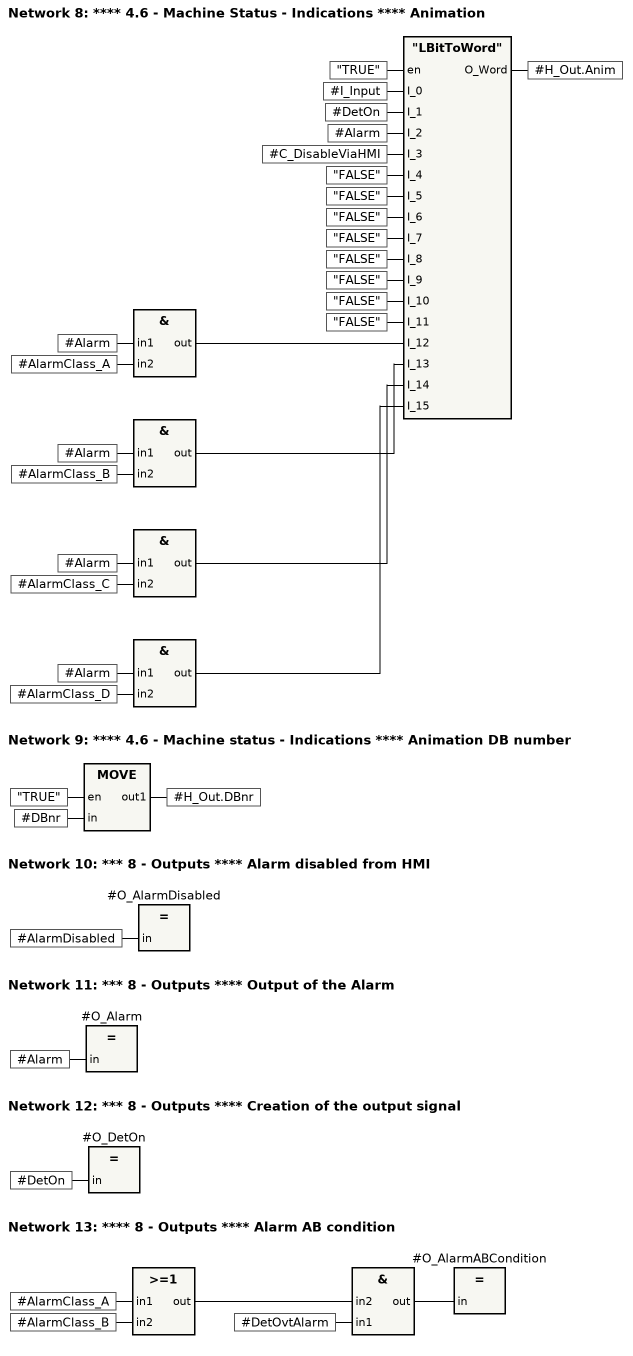
   IF "TRUE" THEN
       "LBitToWord"(I_0 := #I_Input,
                    I_1 := #DetOn,
                    I_2 := #Alarm,
                    I_3 := #C_DisableViaHMI,
                    I_4 := "FALSE",
                    I_5 := "FALSE",
                    I_6 := "FALSE",
                    I_7 := "FALSE",
                    I_8 := "FALSE",
                    I_9 := "FALSE",
                    I_10 := "FALSE",
                    I_11 := "FALSE",
                    I_12 := #Alarm AND #AlarmClass_A,
                    I_13 := #Alarm AND #AlarmClass_B,
                    I_14 := #Alarm AND #AlarmClass_C,
                    I_15 := #Alarm AND #AlarmClass_D,
                    O_Word => #H_Out.Anim);
   END_IF;
END_REGION

REGION Network 9: **** 4.6 - Machine status - Indications **** Animation DB number
   // Animation DB number
   IF "TRUE" THEN #H_Out.DBnr := #DBnr; END_IF;
END_REGION

REGION Network 10: *** 8 - Outputs **** Alarm disabled from HMI
   // Alarm disabled from HMI
   #O_AlarmDisabled := #AlarmDisabled;
END_REGION

REGION Network 11: *** 8 - Outputs **** Output of the Alarm
   // Output of the Alarm
   #O_Alarm := #Alarm;
END_REGION

REGION Network 12: *** 8 - Outputs **** Creation of the output signal
   // Creation of the output signal
   #O_DetOn := #DetOn;
END_REGION

REGION Network 13: **** 8 - Outputs **** Alarm AB condition
   // Alarm AB condition
   #O_AlarmABCondition := (#AlarmClass_A OR #AlarmClass_B) AND #DetOvtAlarm;
END_REGION
END_FUNCTION_BLOCK

FUNCTION_BLOCK "L1SafetyAlarm"   // FB1418, FBD
TITLE = L1SafetyAlarm
{ S7_Optimized_Access := 'FALSE' }
AUTHOR : VCC
FAMILY : AlarmHnd
NAME : 1SafeAlm
VERSION : 0.3
// ================================================================================
// This module is used everywhere one alarm shall be generated when one security 
// input becomes False.
// The alarm can be True only when the input Enable Alarm is also True.
// When the condition to generate the alarm is not fullfilled, a boolean output is 
// available to inform the upper level that the alarm can be reset.
// The alarm is reset by means of the AlarmResetPB signal.
// 
// This module generates also a word containing all necessary information for HMI 
// Icon animation, and a word with all information for HMI safety module 
// diagnostic 
// screen. 
// ================================================================================
// stored: AutoNumber false, IsIECCheckEnabled false, SetENOAutomatically False, UDAEnableTagReadback false
   VAR_INPUT
      I_Input { ExternalAccessible := 'False'; ExternalVisible := 'False'; ExternalWritable := 'False'} : Bool;   // Input safety alarm (normally closed)
      I_AlarmClass { ExternalAccessible := 'False'; ExternalVisible := 'False'; ExternalWritable := 'False'} : Char;   // Alarm class -> A - B - C - D or E
      I_EnableAlarm { ExternalAccessible := 'False'; ExternalVisible := 'False'; ExternalWritable := 'False'} : Bool := TRUE;   // Enable alarm from upper level
      I_AlarmResetPB { ExternalAccessible := 'False'; ExternalVisible := 'False'; ExternalWritable := 'False'} : Bool;   // Alarm reset pushbutton is activated
      I_SafetyCard_PASS_OUT { ExternalAccessible := 'False'; ExternalVisible := 'False'; ExternalWritable := 'False'} : Bool;   // Automatically generated DB from F-Modul (F-Peripherie DB)
      I_SafetyCard_ACK_REQ { ExternalAccessible := 'False'; ExternalVisible := 'False'; ExternalWritable := 'False'} : Bool;   // Automatically generated DB from F-Modul (F-Peripherie DB)
      I_SafetyCard_DIAG { ExternalAccessible := 'False'; ExternalVisible := 'False'; ExternalWritable := 'False'} : Byte;   // Automatically generated DB from F-Modul (F-Peripherie DB)
      I_SafetyCardHWSub { ExternalAccessible := 'False'; ExternalVisible := 'False'; ExternalWritable := 'False'} : HW_SUBMODULE;   // Safety I/O connection hardware
      I_ChannelNr { ExternalAccessible := 'False'; ExternalVisible := 'False'; ExternalWritable := 'False'} : Int;   // Used Channel Nr (Value : 0, 1, 2, 3)
      C_DisableQBadCh { ExternalAccessible := 'False'; ExternalVisible := 'False'; ExternalWritable := 'False'} : Bool;   // Passivation Channel (QbadCh1)
   END_VAR
   VAR_OUTPUT
      O_Alarm { ExternalAccessible := 'False'; ExternalVisible := 'False'; ExternalWritable := 'False'} : Bool;   // Alarm
      O_AlarmABCondition { ExternalAccessible := 'False'; ExternalVisible := 'False'; ExternalWritable := 'False'} : Bool;   // Alarm AB condition
      H_IAnim { ExternalAccessible := 'False'; ExternalVisible := 'False'; ExternalWritable := 'False'} : Word;   // Icon Animation
   END_VAR
   VAR DB_SPECIFIC
      H_Out : Struct   // HMI
         Anim : Word;   // HMI Animation of the object
         DBnr : Int;   // HMI Animation DB number
      END_STRUCT;
      Alarm { ExternalAccessible := 'False'; ExternalVisible := 'False'; ExternalWritable := 'False'} : Bool;   // Alarm
      AlarmClass_A { ExternalAccessible := 'False'; ExternalVisible := 'False'; ExternalWritable := 'False'} : Bool;   // The alarm is from alarm class A
      AlarmClass_B { ExternalAccessible := 'False'; ExternalVisible := 'False'; ExternalWritable := 'False'} : Bool;   // The alarm is from alarm class B
      AlarmClass_C { ExternalAccessible := 'False'; ExternalVisible := 'False'; ExternalWritable := 'False'} : Bool;   // The alarm is from alarm class C
      AlarmClass_D { ExternalAccessible := 'False'; ExternalVisible := 'False'; ExternalWritable := 'False'} : Bool;   // The alarm is from alarm class D
      QbadCh1 { ExternalAccessible := 'False'; ExternalVisible := 'False'; ExternalWritable := 'False'} : Bool;   // Passivation first Channel
      Ack_Req { ExternalAccessible := 'False'; ExternalVisible := 'False'; ExternalWritable := 'False'} : Bool;   // Acknowledgement request
      Timeout_F_I_O { ExternalAccessible := 'False'; ExternalVisible := 'False'; ExternalWritable := 'False'} : Bool;   // Timeout detected by F-I/O
      ChannelFault_F_I_O { ExternalAccessible := 'False'; ExternalVisible := 'False'; ExternalWritable := 'False'} : Bool;   // F-I/O fault or channel fault detected by F-I/O
      CRCSeqError_F_I_O { ExternalAccessible := 'False'; ExternalVisible := 'False'; ExternalWritable := 'False'} : Bool;   // CRC error or sequence number error detected by F-I/O
      Timeout_F_Sys { ExternalAccessible := 'False'; ExternalVisible := 'False'; ExternalWritable := 'False'} : Bool;   // Timeout detected by F-System
      SeqError_F_Sys { ExternalAccessible := 'False'; ExternalVisible := 'False'; ExternalWritable := 'False'} : Bool;   // Sequence number error detected by F-system
      CRCError_F_Sys { ExternalAccessible := 'False'; ExternalVisible := 'False'; ExternalWritable := 'False'} : Bool;   // CRC error detected by F-system
      AlarmCond { ExternalAccessible := 'False'; ExternalVisible := 'False'; ExternalWritable := 'False'} : Bool;   // Alarm condition
      RetValueData { ExternalAccessible := 'False'; ExternalVisible := 'False'; ExternalWritable := 'False'} : Int;   // Status variable (SFC14)
      DBnr { ExternalAccessible := 'False'; ExternalVisible := 'False'; ExternalWritable := 'False'} : Int;   // HMI DB number
   END_VAR
   VAR_TEMP
      T_DataFromSafetyCard : Struct   // Temp structure : receive data's from Safety Card
         Byte0_Bit0_Spare : Bool;
         Byte0_Bit1_Spare : Bool;
         Byte0_Bit2_Spare : Bool;
         Byte0_Bit3_Spare : Bool;
         Byte0_Bit4_Spare : Bool;
         Byte0_Bit5_Spare : Bool;
         Byte0_Bit6_Spare : Bool;
         Byte0_Bit7_Spare : Bool;
         Byte1_Bit0_QBadCh0 : Bool;
         Byte1_Bit1_QBadCh1 : Bool;
         Byte1_Bit2_QBadCh2 : Bool;
         Byte1_Bit3_QBadCh3 : Bool;
         Byte1_Bit4_QBadCh4 : Bool;
         Byte1_Bit5_QBadCh5 : Bool;
         Byte1_Bit6_QBadCh6 : Bool;
         Byte1_Bit7_QBadCh7 : Bool;
         Byte2_bit0_Spare : Bool;
         Byte2_bit1_Spare : Bool;
         Byte2_bit2_Spare : Bool;
         Byte2_bit3_Spare : Bool;
         Byte2_bit4_Spare : Bool;
         Byte2_bit5_Spare : Bool;
         Byte2_bit6_Spare : Bool;
         Byte2_bit7_Spare : Bool;
         Byte3_Bit0_Spare : Bool;
         Byte3_Bit1_Spare : Bool;
         Byte3_Bit2_Spare : Bool;
         Byte3_Bit3_Spare : Bool;
         Byte3_Bit4_Spare : Bool;
         Byte3_Bit5_Spare : Bool;
         Byte3_Bit6_Spare : Bool;
         Byte3_Bit7_Spare : Bool;
         Byte4_bit0_Spare : Bool;
         Byte4_bit1_Spare : Bool;
         Byte4_bit2_Spare : Bool;
         Byte4_bit3_Spare : Bool;
         Byte4_bit4_Spare : Bool;
         Byte4_bit5_Spare : Bool;
         Byte4_bit6_Spare : Bool;
         Byte4_bit7_Spare : Bool;
         Byte5_bit0_Spare : Bool;
         Byte5_bit1_Spare : Bool;
         Byte5_bit2_Spare : Bool;
         Byte5_bit3_Spare : Bool;
         Byte5_bit4_Spare : Bool;
         Byte5_bit5_Spare : Bool;
         Byte5_bit6_Spare : Bool;
         Byte5_bit7_Spare : Bool;
      END_STRUCT;
   END_VAR
BEGIN

NETWORK
TITLE = **** 1 - Inputs **** DB number
// DB number
      L     DINO;
      T     #DBnr;

NETWORK
TITLE = **** 1 - Inputs **** Alarm class
// Alarm class
// Alarm class = D
      L     #I_AlarmClass;
      L     'D';
      ==I;
      =     #AlarmClass_D;

// Alarm class = C
      L     #I_AlarmClass;
      L     'C';
      ==I;
      =     #AlarmClass_C;

// Alarm class = B
      L     #I_AlarmClass;
      L     'B';
      ==I;
      =     #AlarmClass_B;

// Alarm class = A
      AN    #AlarmClass_B;
      AN    #AlarmClass_C;
      AN    #AlarmClass_D;
      =     #AlarmClass_A;


REGION Network 3: **** 1 - Inputs **** Safety I/O connection hardware
   // Safety I/O connection hardware
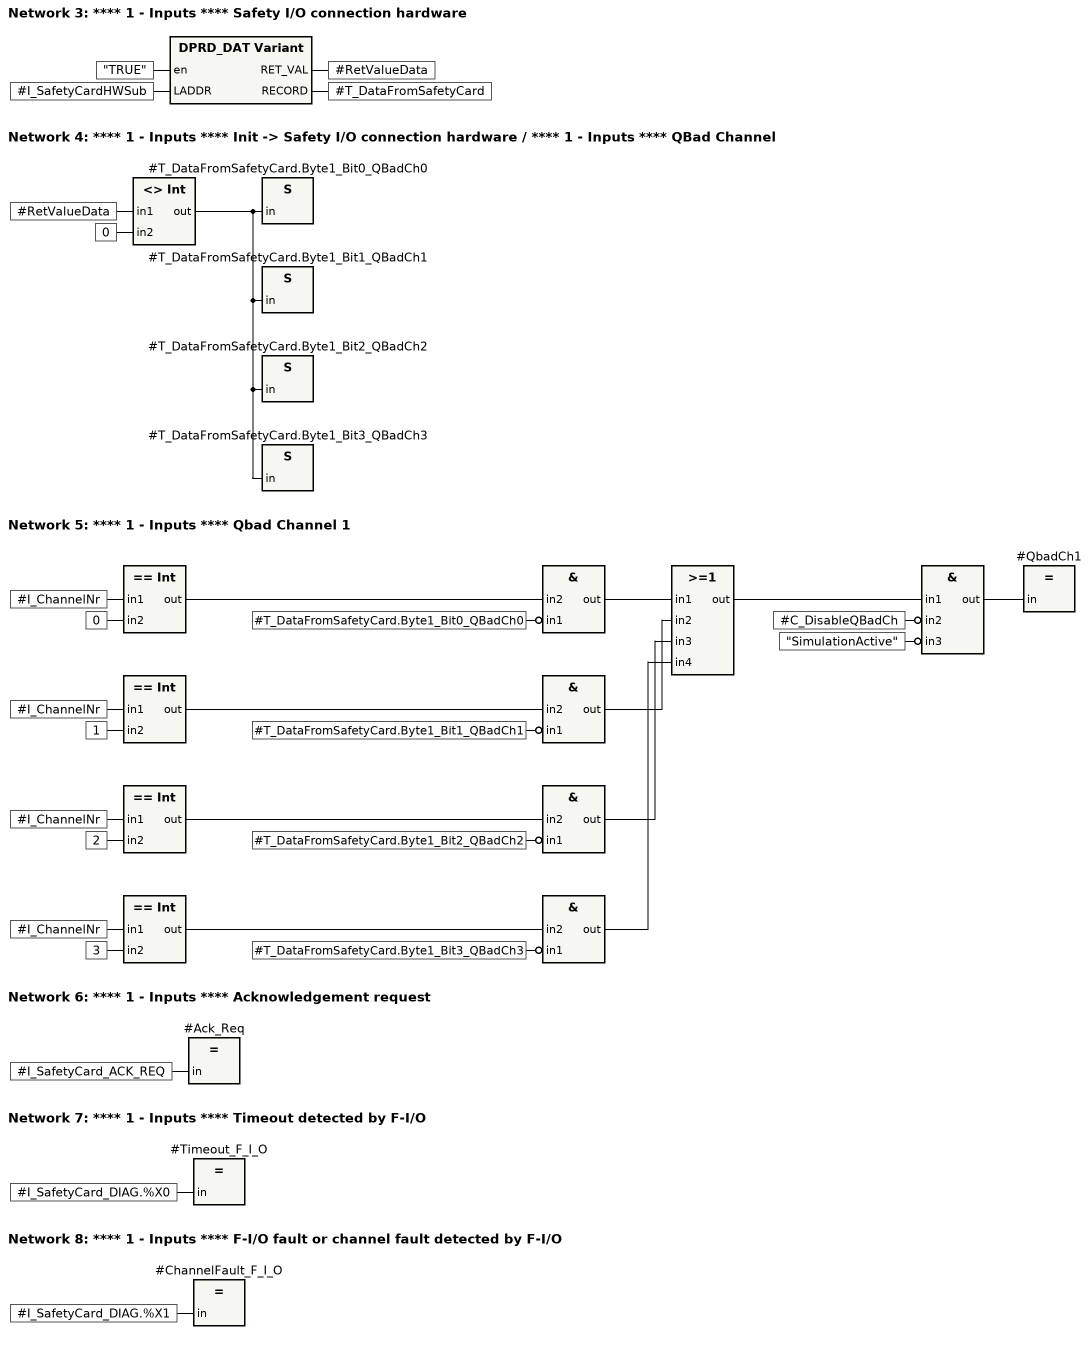
   IF "TRUE" THEN
       #RetValueData := DPRD_DAT(LADDR := #I_SafetyCardHWSub, RECORD => #T_DataFromSafetyCard);
   END_IF;
END_REGION

REGION Network 4: **** 1 - Inputs **** Init -> Safety I/O connection hardware / **** 1 - Inputs **** QBad Channel
   // Init -> Safety I/O connection hardware
   IF #RetValueData <> 0 THEN
       #T_DataFromSafetyCard.Byte1_Bit0_QBadCh0 := TRUE;
       #T_DataFromSafetyCard.Byte1_Bit1_QBadCh1 := TRUE;
       #T_DataFromSafetyCard.Byte1_Bit2_QBadCh2 := TRUE;
       #T_DataFromSafetyCard.Byte1_Bit3_QBadCh3 := TRUE;
   END_IF;
END_REGION

REGION Network 5: **** 1 - Inputs **** Qbad Channel 1
   // Qbad Channel 1
   #QbadCh1 := (((#I_ChannelNr = 0) AND NOT #T_DataFromSafetyCard.Byte1_Bit0_QBadCh0) OR ((#I_ChannelNr = 1) AND NOT #T_DataFromSafetyCard.Byte1_Bit1_QBadCh1) OR ((#I_ChannelNr = 2) AND NOT #T_DataFromSafetyCard.Byte1_Bit2_QBadCh2) OR ((#I_ChannelNr = 3) AND NOT #T_DataFromSafetyCard.Byte1_Bit3_QBadCh3)) AND NOT #C_DisableQBadCh AND NOT "SimulationActive";
END_REGION

REGION Network 6: **** 1 - Inputs **** Acknowledgement request
   // Acknowledgement request
   #Ack_Req := #I_SafetyCard_ACK_REQ;
END_REGION

REGION Network 7: **** 1 - Inputs **** Timeout detected by F-I/O
   // Timeout detected by F-I/O
   #Timeout_F_I_O := #I_SafetyCard_DIAG.%X0;
END_REGION

REGION Network 8: **** 1 - Inputs **** F-I/O fault or channel fault detected by F-I/O
   // F-I/O fault or channel fault detected by F-I/O
   #ChannelFault_F_I_O := #I_SafetyCard_DIAG.%X1;
END_REGION

REGION Network 9: **** 1 - Inputs **** CRC error or sequence number error detected by F-I/O
   // CRC error or sequence number error detected by F-I/O
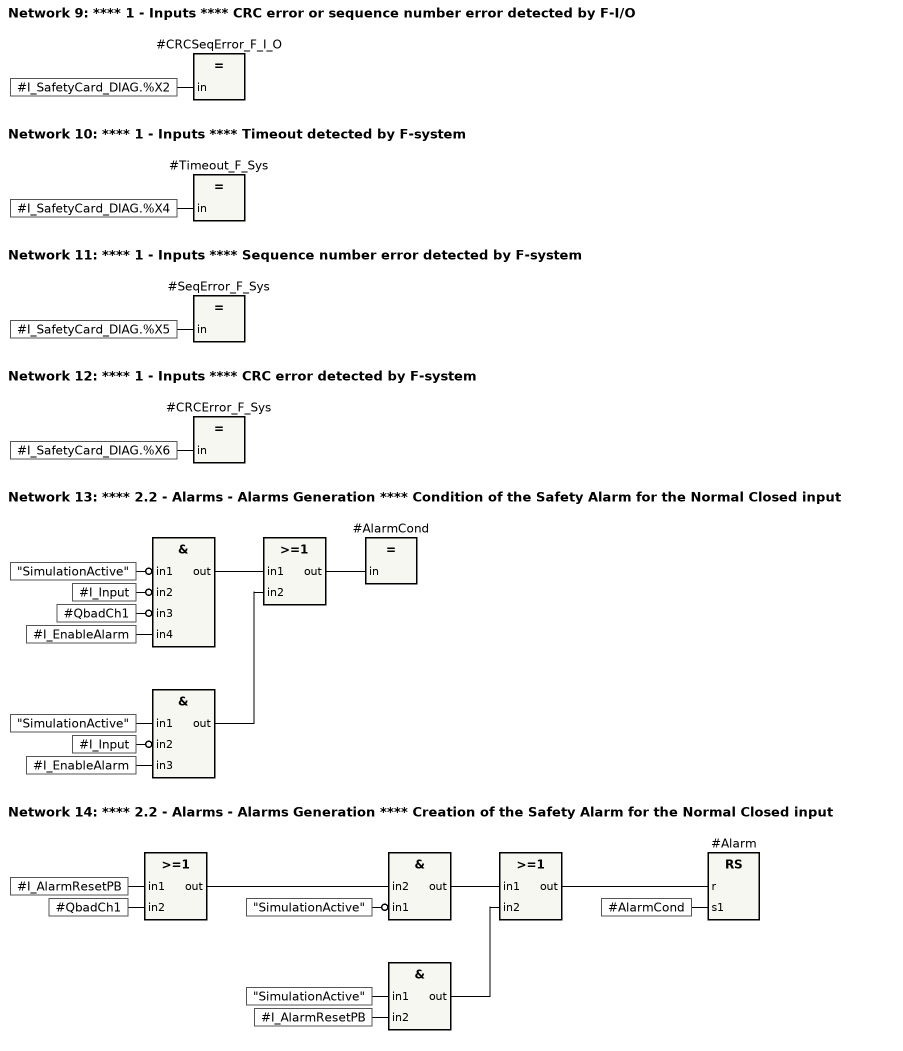
   #CRCSeqError_F_I_O := #I_SafetyCard_DIAG.%X2;
END_REGION

REGION Network 10: **** 1 - Inputs **** Timeout detected by F-system
   // Timeout detected by F-system
   #Timeout_F_Sys := #I_SafetyCard_DIAG.%X4;
END_REGION

REGION Network 11: **** 1 - Inputs **** Sequence number error detected by F-system
   // Sequence number error detected by F-system
   #SeqError_F_Sys := #I_SafetyCard_DIAG.%X5;
END_REGION

REGION Network 12: **** 1 - Inputs **** CRC error detected by F-system
   // CRC error detected by F-system
   #CRCError_F_Sys := #I_SafetyCard_DIAG.%X6;
END_REGION

REGION Network 13: **** 2.2 - Alarms - Alarms Generation **** Condition of the Safety Alarm for the Normal Closed input
   // Condition of the Safety Alarm for the Normal Closed input
   #AlarmCond := (NOT "SimulationActive" AND NOT #I_Input AND NOT #QbadCh1 AND #I_EnableAlarm) OR ("SimulationActive" AND NOT #I_Input AND #I_EnableAlarm);
END_REGION

REGION Network 14: **** 2.2 - Alarms - Alarms Generation **** Creation of the Safety Alarm for the Normal Closed input
   // Creation of the Safety Alarm for the Normal Closed input
   IF ((#I_AlarmResetPB OR #QbadCh1) AND NOT "SimulationActive") OR ("SimulationActive" AND #I_AlarmResetPB) THEN
       #Alarm := FALSE;   // RS flip-flop
   END_IF;
   IF #AlarmCond THEN #Alarm := TRUE; END_IF;
END_REGION

REGION Network 15: **** 4.6 - Machine Status - Indications **** Icon Animation
   // Icon Animation
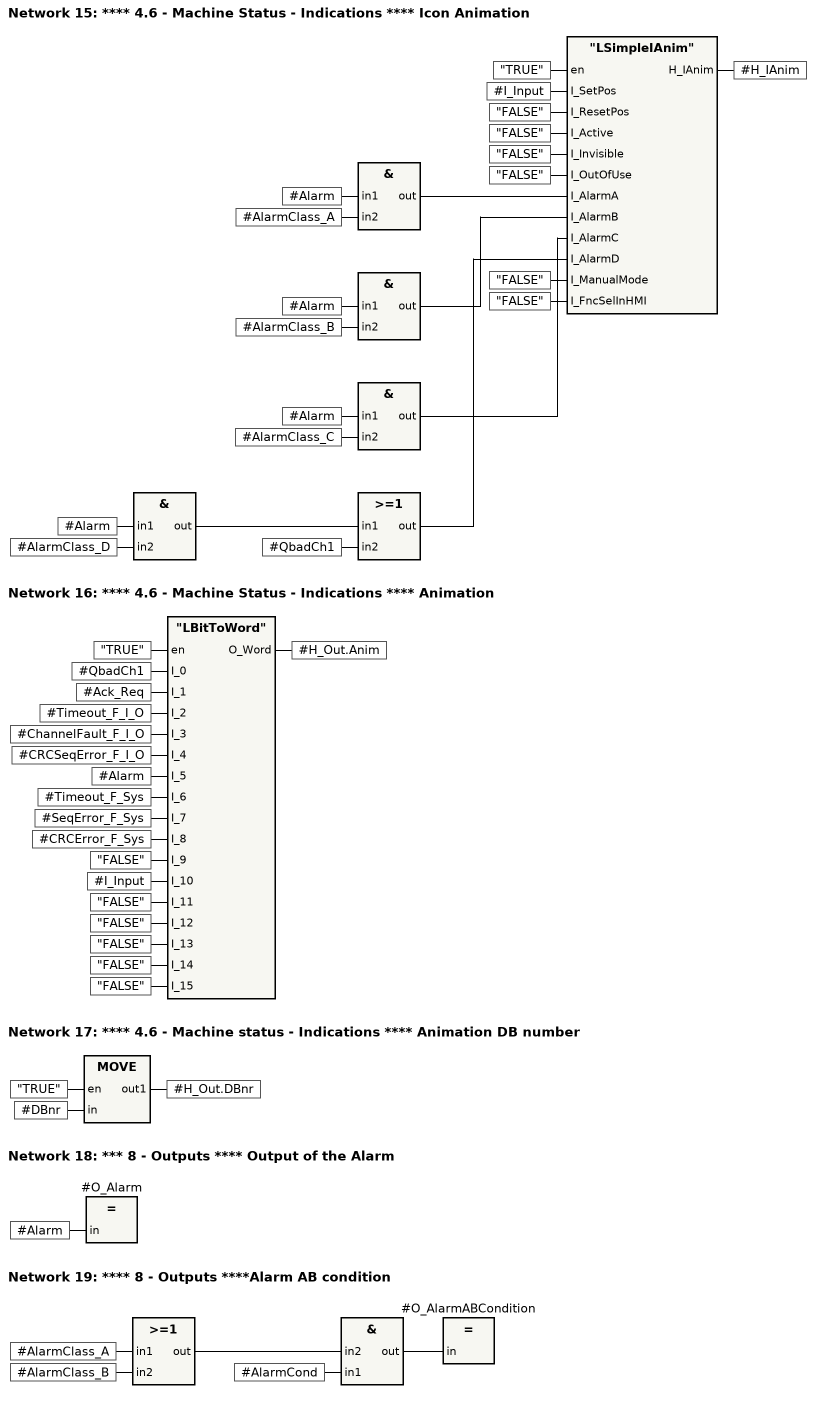
   IF "TRUE" THEN
       "LSimpleIAnim"(I_SetPos := #I_Input,
                      I_ResetPos := "FALSE",
                      I_Active := "FALSE",
                      I_Invisible := "FALSE",
                      I_OutOfUse := "FALSE",
                      I_AlarmA := #Alarm AND #AlarmClass_A,
                      I_AlarmB := #Alarm AND #AlarmClass_B,
                      I_AlarmC := #Alarm AND #AlarmClass_C,
                      I_AlarmD := (#Alarm AND #AlarmClass_D) OR #QbadCh1,
                      I_ManualMode := "FALSE",
                      I_FncSelInHMI := "FALSE",
                      H_IAnim => #H_IAnim);
   END_IF;
END_REGION

REGION Network 16: **** 4.6 - Machine Status - Indications **** Animation
   // Animation
   IF "TRUE" THEN
       "LBitToWord"(I_0 := #QbadCh1,
                    I_1 := #Ack_Req,
                    I_2 := #Timeout_F_I_O,
                    I_3 := #ChannelFault_F_I_O,
                    I_4 := #CRCSeqError_F_I_O,
                    I_5 := #Alarm,
                    I_6 := #Timeout_F_Sys,
                    I_7 := #SeqError_F_Sys,
                    I_8 := #CRCError_F_Sys,
                    I_9 := "FALSE",
                    I_10 := #I_Input,
                    I_11 := "FALSE",
                    I_12 := "FALSE",
                    I_13 := "FALSE",
                    I_14 := "FALSE",
                    I_15 := "FALSE",
                    O_Word => #H_Out.Anim);
   END_IF;
END_REGION

REGION Network 17: **** 4.6 - Machine status - Indications **** Animation DB number
   // Animation DB number
   IF "TRUE" THEN #H_Out.DBnr := #DBnr; END_IF;
END_REGION

REGION Network 18: *** 8 - Outputs **** Output of the Alarm
   // Output of the Alarm
   #O_Alarm := #Alarm;
END_REGION

REGION Network 19: **** 8 - Outputs ****Alarm AB condition
   // Alarm AB condition
   #O_AlarmABCondition := (#AlarmClass_A OR #AlarmClass_B) AND #AlarmCond;
END_REGION
END_FUNCTION_BLOCK

FUNCTION_BLOCK "LRedundantDet"   // FB1419, FBD
TITLE = LRedundantDet
{ S7_Optimized_Access := 'FALSE' }
AUTHOR : VCC
FAMILY : AlarmHnd
NAME : RedunDet
VERSION : 1.0
// ================================================================================
// This module is used everywhere 2 redundant detections are needed on working 
// area to avoid activation with safety shoes.
// If the alarm is enable, one alarm shall be generated
// when detection 1 is true and some time later the detection 2 is still false
// or when detection 2 is true and some time later the detection 1 is still false
// then Alarm is generated.
// Alarm is disable from HMI, a boolean output is available to inform the upper 
// level and do action in the Alarm summary.
// When the conditions to generate the alarm is disappear, a boolean output is 
// available to inform the upper level that the alarm can be reset.
// The alarm is reset by means of the AlarmResetPB signal.
// ================================================================================
// stored: AutoNumber false, IsIECCheckEnabled false, SetENOAutomatically False, UDAEnableTagReadback false
   VAR_INPUT
      I_Detection1 { ExternalAccessible := 'False'; ExternalVisible := 'False'; ExternalWritable := 'False'} : Bool;   // Input signal of detection 1
      I_Detection2 { ExternalAccessible := 'False'; ExternalVisible := 'False'; ExternalWritable := 'False'} : Bool;   // Input signal of detection 2
      I_EnableAlarm { ExternalAccessible := 'False'; ExternalVisible := 'False'; ExternalWritable := 'False'} : Bool := TRUE;   // Enable alarm from upper level
      I_Invisible { ExternalAccessible := 'False'; ExternalVisible := 'False'; ExternalWritable := 'False'} : Bool;   // Invisible
      I_AlarmResetPB { ExternalAccessible := 'False'; ExternalVisible := 'False'; ExternalWritable := 'False'} : Bool;   // Alarm reset pushbutton is activated
      I_TimeDelay { ExternalAccessible := 'False'; ExternalVisible := 'False'; ExternalWritable := 'False'} : DInt;   // Time delay value (1 unit = 1 ms)
      H_In : Struct   // HMI
         DisableAlarm : Bool;   // Disable alarm from HMI
      END_STRUCT;
   END_VAR
   VAR_OUTPUT
      O_RedundantDetAlm { ExternalAccessible := 'False'; ExternalVisible := 'False'; ExternalWritable := 'False'} : Bool;   // Redundant detection Alarm
      O_AlarmDisabled { ExternalAccessible := 'False'; ExternalVisible := 'False'; ExternalWritable := 'False'} : Bool;   // Alarm disabled from HMI
      O_AlarmABCondition { ExternalAccessible := 'False'; ExternalVisible := 'False'; ExternalWritable := 'False'} : Bool;   // Alarm AB condition
      H_IAnim { ExternalAccessible := 'False'; ExternalVisible := 'False'; ExternalWritable := 'False'} : Word;
      H_Out : Struct   // HMI
         Anim : Word;   // HMI Animation of the object
      END_STRUCT;
   END_VAR
   VAR DB_SPECIFIC
      DelayTimeResult { ExternalAccessible := 'False'; ExternalVisible := 'False'; ExternalWritable := 'False'} : Bool;   // Delay time boolean
      Detection1Mem { ExternalAccessible := 'False'; ExternalVisible := 'False'; ExternalWritable := 'False'} : Bool;   // Memory detyection 1 on true
      Detection2Mem { ExternalAccessible := 'False'; ExternalVisible := 'False'; ExternalWritable := 'False'} : Bool;   // Memory detyection 2 on true
      ResetDetectionMem { ExternalAccessible := 'False'; ExternalVisible := 'False'; ExternalWritable := 'False'} : Bool;   // condition to reset the detection memories
      SummaryRedundantDetAlm { ExternalAccessible := 'False'; ExternalVisible := 'False'; ExternalWritable := 'False'} : Bool;   // Summary redundant detection Alarm
      RedundantDetAlm { ExternalAccessible := 'False'; ExternalVisible := 'False'; ExternalWritable := 'False'} : Bool;   // Redundant detection Alarm
      RedundantDetAlmCond { ExternalAccessible := 'False'; ExternalVisible := 'False'; ExternalWritable := 'False'} : Bool;   // Redundant detection Alarm condition
   END_VAR
   VAR
      DelayTimer { ExternalAccessible := 'False'; ExternalVisible := 'False'; ExternalWritable := 'False'; S7_SetPoint := 'True'} : "LTimer";
   END_VAR
BEGIN

REGION Network 1: **** 2.2 - Alarms - Alarms Generation **** Creation of delay time
   // Creation of delay time
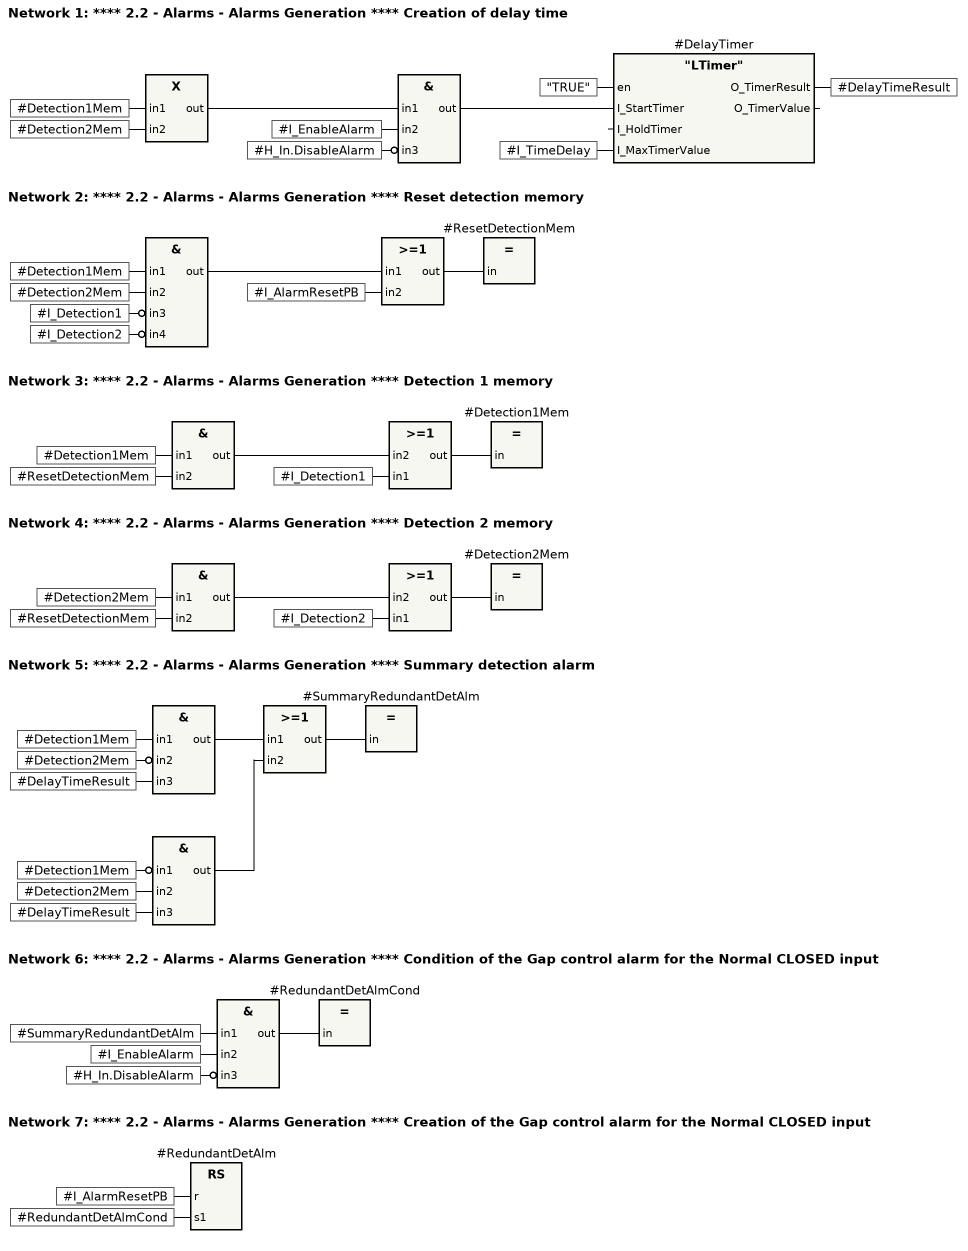
   IF "TRUE" THEN
       #DelayTimer(I_StartTimer := (#Detection1Mem XOR #Detection2Mem) AND #I_EnableAlarm AND NOT #H_In.DisableAlarm,   // "LTimer"
                   I_MaxTimerValue := #I_TimeDelay,
                   O_TimerResult => #DelayTimeResult);
   END_IF;
END_REGION

REGION Network 2: **** 2.2 - Alarms - Alarms Generation **** Reset detection memory
   // Reset detection memory
   #ResetDetectionMem := (#Detection1Mem AND #Detection2Mem AND NOT #I_Detection1 AND NOT #I_Detection2) OR #I_AlarmResetPB;
END_REGION

REGION Network 3: **** 2.2 - Alarms - Alarms Generation **** Detection 1 memory
   // Detection 1 memory
   #Detection1Mem := (#Detection1Mem AND #ResetDetectionMem) OR #I_Detection1;
END_REGION

REGION Network 4: **** 2.2 - Alarms - Alarms Generation **** Detection 2 memory
   // Detection 2 memory
   #Detection2Mem := (#Detection2Mem AND #ResetDetectionMem) OR #I_Detection2;
END_REGION

REGION Network 5: **** 2.2 - Alarms - Alarms Generation **** Summary detection alarm
   // Summary detection alarm
   #SummaryRedundantDetAlm := (#Detection1Mem AND NOT #Detection2Mem AND #DelayTimeResult) OR (NOT #Detection1Mem AND #Detection2Mem AND #DelayTimeResult);
END_REGION

REGION Network 6: **** 2.2 - Alarms - Alarms Generation **** Condition of the Gap control alarm for the Normal CLOSED input
   // Condition of the Gap control alarm for the Normal CLOSED input
   #RedundantDetAlmCond := #SummaryRedundantDetAlm AND #I_EnableAlarm AND NOT #H_In.DisableAlarm;
END_REGION

REGION Network 7: **** 2.2 - Alarms - Alarms Generation **** Creation of the Gap control alarm for the Normal CLOSED input
   // Creation of the Gap control alarm for the Normal CLOSED input
   IF #I_AlarmResetPB THEN
       #RedundantDetAlm := FALSE;   // RS flip-flop
   END_IF;
   IF #RedundantDetAlmCond THEN #RedundantDetAlm := TRUE; END_IF;
END_REGION

REGION Network 8: **** 4.6 - Mashine Status - Indications **** Icon Animation
   // Icon Animation
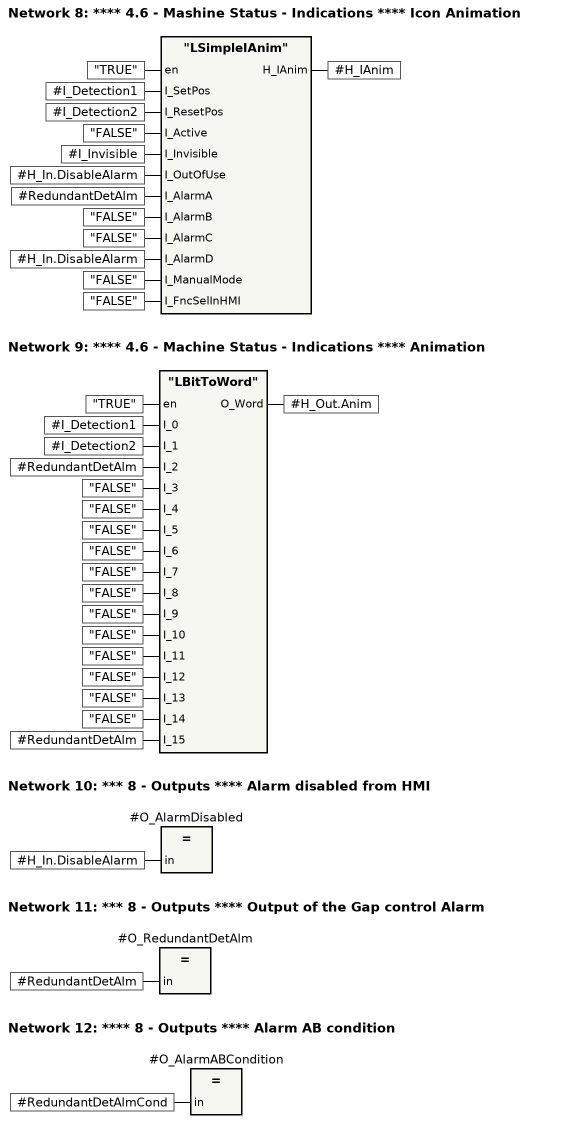
   IF "TRUE" THEN
       "LSimpleIAnim"(I_SetPos := #I_Detection1,
                      I_ResetPos := #I_Detection2,
                      I_Active := "FALSE",
                      I_Invisible := #I_Invisible,
                      I_OutOfUse := #H_In.DisableAlarm,
                      I_AlarmA := #RedundantDetAlm,
                      I_AlarmB := "FALSE",
                      I_AlarmC := "FALSE",
                      I_AlarmD := #H_In.DisableAlarm,
                      I_ManualMode := "FALSE",
                      I_FncSelInHMI := "FALSE",
                      H_IAnim => #H_IAnim);
   END_IF;
END_REGION

REGION Network 9: **** 4.6 - Machine Status - Indications **** Animation
   // Animation
   IF "TRUE" THEN
       "LBitToWord"(I_0 := #I_Detection1,
                    I_1 := #I_Detection2,
                    I_2 := #RedundantDetAlm,
                    I_3 := "FALSE",
                    I_4 := "FALSE",
                    I_5 := "FALSE",
                    I_6 := "FALSE",
                    I_7 := "FALSE",
                    I_8 := "FALSE",
                    I_9 := "FALSE",
                    I_10 := "FALSE",
                    I_11 := "FALSE",
                    I_12 := "FALSE",
                    I_13 := "FALSE",
                    I_14 := "FALSE",
                    I_15 := #RedundantDetAlm,
                    O_Word => #H_Out.Anim);
   END_IF;
END_REGION

REGION Network 10: *** 8 - Outputs **** Alarm disabled from HMI
   // Alarm disabled from HMI
   #O_AlarmDisabled := #H_In.DisableAlarm;
END_REGION

REGION Network 11: *** 8 - Outputs **** Output of the Gap control Alarm
   // Output of the Gap control Alarm
   #O_RedundantDetAlm := #RedundantDetAlm;
END_REGION

REGION Network 12: **** 8 - Outputs **** Alarm AB condition
   // Alarm AB condition
   #O_AlarmABCondition := #RedundantDetAlmCond;
END_REGION
END_FUNCTION_BLOCK

FUNCTION_BLOCK "LPassivate"   // FB1420, FBD
TITLE = LPassivate
{ S7_Optimized_Access := 'FALSE' }
AUTHOR : VCC
FAMILY : AlarmHnd
NAME : Passivat
VERSION : 0.1
// ================================================================================
// This module is used everywhere passivation of a slot shall generate an alarm.
// The alarm can be True only when the input Enable Alarm is also True.
// When the condition to generate the alarm is not fullfilled, a boolean output is 
// available to inform the upper level that the alarm can be reset.
// The alarm is reset by means of the AlarmResetPB signal.
// ================================================================================
// stored: AutoNumber false, IsIECCheckEnabled false, SetENOAutomatically False, UDAEnableTagReadback false
   VAR_INPUT
      I_SafetyCard_PASS_OUT { ExternalAccessible := 'False'; ExternalVisible := 'False'; ExternalWritable := 'False'} : Bool;   // Automatically generated DB from F-Modul (F-Peripherie DB)
      I_SafetyCard_ACK_REQ { ExternalAccessible := 'False'; ExternalVisible := 'False'; ExternalWritable := 'False'} : Bool;   // Automatically generated DB from F-Modul (F-Peripherie DB)
      I_SafetyCard_DIAG { ExternalAccessible := 'False'; ExternalVisible := 'False'; ExternalWritable := 'False'} : Byte;   // Automatically generated DB from F-Modul (F-Peripherie DB)
      I_SafetyCardHWSub { ExternalAccessible := 'False'; ExternalVisible := 'False'; ExternalWritable := 'False'} : HW_SUBMODULE;   // Safety I/O connection hardware
      I_AlarmClass { ExternalAccessible := 'False'; ExternalVisible := 'False'; ExternalWritable := 'False'} : Char;   // Alarm class -> A - B - C - D or E
      I_EnableAlarm { ExternalAccessible := 'False'; ExternalVisible := 'False'; ExternalWritable := 'False'} : Bool := TRUE;   // Enable alarm from upper level
      I_AlarmResetPB { ExternalAccessible := 'False'; ExternalVisible := 'False'; ExternalWritable := 'False'} : Bool;   // Alarm reset pushbutton is activated
      C_OutputCard { ExternalAccessible := 'False'; ExternalVisible := 'False'; ExternalWritable := 'False'} : Bool;   // 1 = The safety card is an output card
   END_VAR
   VAR_OUTPUT
      O_PassivateAlm { ExternalAccessible := 'False'; ExternalVisible := 'False'; ExternalWritable := 'False'} : Bool;   // Alarm
      O_AlarmABCondition { ExternalAccessible := 'False'; ExternalVisible := 'False'; ExternalWritable := 'False'} : Bool;   // Alarm AB condition
      H_IAnim { ExternalAccessible := 'False'; ExternalVisible := 'False'; ExternalWritable := 'False'} : Word;   // Icon animation
   END_VAR
   VAR DB_SPECIFIC
      H_Out : Struct   // HMI
         Anim : Word;   // HMI Animation of the object
         DBnr : Int;   // HMI Animation DB number
      END_STRUCT;
      Alarm { ExternalAccessible := 'False'; ExternalVisible := 'False'; ExternalWritable := 'False'} : Bool;   // Alarm
      AlarmClass_A { ExternalAccessible := 'False'; ExternalVisible := 'False'; ExternalWritable := 'False'} : Bool;   // The alarm is from alarm class A
      AlarmClass_B { ExternalAccessible := 'False'; ExternalVisible := 'False'; ExternalWritable := 'False'} : Bool;   // The alarm is from alarm class B
      AlarmClass_C { ExternalAccessible := 'False'; ExternalVisible := 'False'; ExternalWritable := 'False'} : Bool;   // The alarm is from alarm class C
      AlarmClass_D { ExternalAccessible := 'False'; ExternalVisible := 'False'; ExternalWritable := 'False'} : Bool;   // The alarm is from alarm class D
      AlarmCond { ExternalAccessible := 'False'; ExternalVisible := 'False'; ExternalWritable := 'False'} : Bool;   // Alarm condition
      QbadCh0 { ExternalAccessible := 'False'; ExternalVisible := 'False'; ExternalWritable := 'False'} : Bool;   // Passivation first Channel
      QbadCh1 { ExternalAccessible := 'False'; ExternalVisible := 'False'; ExternalWritable := 'False'} : Bool;   // Passivation second Channel
      QbadCh2 { ExternalAccessible := 'False'; ExternalVisible := 'False'; ExternalWritable := 'False'} : Bool;   // Passivation third Channel
      QbadCh3 { ExternalAccessible := 'False'; ExternalVisible := 'False'; ExternalWritable := 'False'} : Bool;   // Passivation fourth Channel
      Ack_Req { ExternalAccessible := 'False'; ExternalVisible := 'False'; ExternalWritable := 'False'} : Bool;   // Acknowledgement request
      Pass_Out { ExternalAccessible := 'False'; ExternalVisible := 'False'; ExternalWritable := 'False'} : Bool;   // Slot is passivated
      Timeout_F_I_O { ExternalAccessible := 'False'; ExternalVisible := 'False'; ExternalWritable := 'False'} : Bool;   // Timeout detected by F-I/O
      ChannelFault_F_I_O { ExternalAccessible := 'False'; ExternalVisible := 'False'; ExternalWritable := 'False'} : Bool;   // F-I/O fault or channel fault detected by F-I/O
      CRCSeqError_F_I_O { ExternalAccessible := 'False'; ExternalVisible := 'False'; ExternalWritable := 'False'} : Bool;   // CRC error or sequence number error detected by F-I/O
      Timeout_F_Sys { ExternalAccessible := 'False'; ExternalVisible := 'False'; ExternalWritable := 'False'} : Bool;   // Timeout detected by F-System
      SeqError_F_Sys { ExternalAccessible := 'False'; ExternalVisible := 'False'; ExternalWritable := 'False'} : Bool;   // Sequence number error detected by F-system
      CRCError_F_Sys { ExternalAccessible := 'False'; ExternalVisible := 'False'; ExternalWritable := 'False'} : Bool;   // CRC error detected by F-system
      RetValueData { ExternalAccessible := 'False'; ExternalVisible := 'False'; ExternalWritable := 'False'} : Int;   // Status variable (SFC14)
      DBnr { ExternalAccessible := 'False'; ExternalVisible := 'False'; ExternalWritable := 'False'} : Int;   // HMI DB number
   END_VAR
   VAR_TEMP
      T_DataFromSafetyCard : Struct   // Temp structure : receive data's from Safety Card
         Byte0_Bit0_QBadCh0 : Bool;
         Byte0_Bit1_QBadCh1 : Bool;
         Byte0_Bit2_QBadCh2 : Bool;
         Byte0_Bit3_QBadCh3 : Bool;
         Byte0_Bit4_Spare : Bool;
         Byte0_Bit5_Spare : Bool;
         Byte0_Bit6_Spare : Bool;
         Byte0_Bit7_Spare : Bool;
         Byte1_Bit0_QBadCh0 : Bool;
         Byte1_Bit1_QBadCh1 : Bool;
         Byte1_Bit2_QBadCh2 : Bool;
         Byte1_Bit3_QBadCh3 : Bool;
         Byte1_Bit4_Spare : Bool;
         Byte1_Bit5_Spare : Bool;
         Byte1_Bit6_Spare : Bool;
         Byte1_Bit7_Spare : Bool;
         Byte2_bit0_Spare : Bool;
         Byte2_bit1_Spare : Bool;
         Byte2_bit2_Spare : Bool;
         Byte2_bit3_Spare : Bool;
         Byte2_bit4_Spare : Bool;
         Byte2_bit5_Spare : Bool;
         Byte2_bit6_Spare : Bool;
         Byte2_bit7_Spare : Bool;
         Byte3_Bit0_Spare : Bool;
         Byte3_Bit1_Spare : Bool;
         Byte3_Bit2_Spare : Bool;
         Byte3_Bit3_Spare : Bool;
         Byte3_Bit4_Spare : Bool;
         Byte3_Bit5_Spare : Bool;
         Byte3_Bit6_Spare : Bool;
         Byte3_Bit7_Spare : Bool;
         Byte4_bit0_Spare : Bool;
         Byte4_bit1_Spare : Bool;
         Byte4_bit2_Spare : Bool;
         Byte4_bit3_Spare : Bool;
         Byte4_bit4_Spare : Bool;
         Byte4_bit5_Spare : Bool;
         Byte4_bit6_Spare : Bool;
         Byte4_bit7_Spare : Bool;
         Byte5_bit0_Spare : Bool;
         Byte5_bit1_Spare : Bool;
         Byte5_bit2_Spare : Bool;
         Byte5_bit3_Spare : Bool;
         Byte5_bit4_Spare : Bool;
         Byte5_bit5_Spare : Bool;
         Byte5_bit6_Spare : Bool;
         Byte5_bit7_Spare : Bool;
      END_STRUCT;
   END_VAR
BEGIN

NETWORK
TITLE = **** 1 - Inputs **** DB number
// DB number
      L     DINO;
      T     #DBnr;

NETWORK
TITLE = **** 1 - Inputs **** Alarm class
// Alarm class
// Alarm class = D
      L     #I_AlarmClass;
      L     'D';
      ==I;
      =     #AlarmClass_D;

// Alarm class = C
      L     #I_AlarmClass;
      L     'C';
      ==I;
      =     #AlarmClass_C;

// Alarm class = B
      L     #I_AlarmClass;
      L     'B';
      ==I;
      =     #AlarmClass_B;

// Alarm class = A
      AN    #AlarmClass_B;
      AN    #AlarmClass_C;
      AN    #AlarmClass_D;
      =     #AlarmClass_A;


REGION Network 3: **** 1 - Inputs **** Safety I/O connection hardware
   // Safety I/O connection hardware
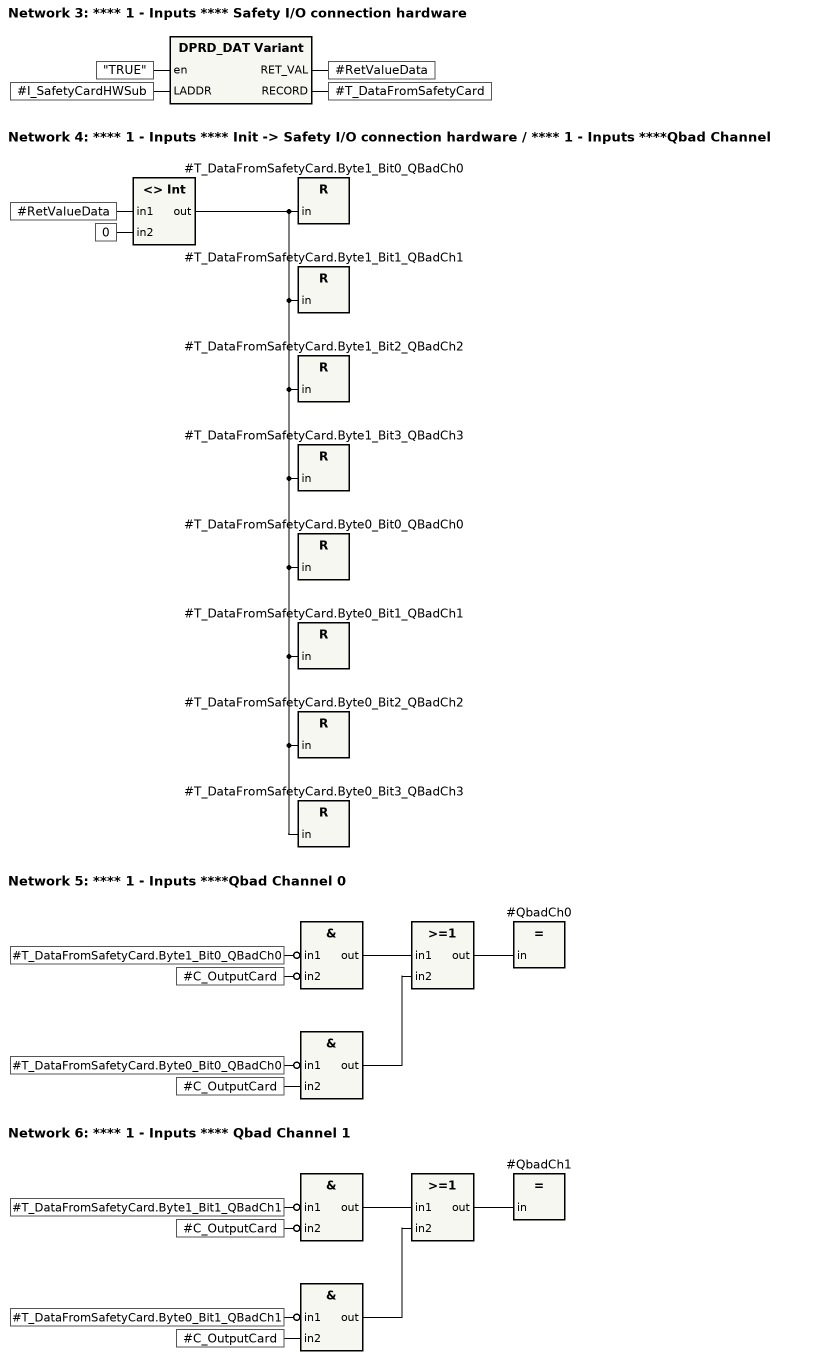
   IF "TRUE" THEN
       #RetValueData := DPRD_DAT(LADDR := #I_SafetyCardHWSub, RECORD => #T_DataFromSafetyCard);
   END_IF;
END_REGION

REGION Network 4: **** 1 - Inputs **** Init -> Safety I/O connection hardware / **** 1 - Inputs ****Qbad Channel
   // Init -> Safety I/O connection hardware
   IF #RetValueData <> 0 THEN
       #T_DataFromSafetyCard.Byte1_Bit0_QBadCh0 := FALSE;
       #T_DataFromSafetyCard.Byte1_Bit1_QBadCh1 := FALSE;
       #T_DataFromSafetyCard.Byte1_Bit2_QBadCh2 := FALSE;
       #T_DataFromSafetyCard.Byte1_Bit3_QBadCh3 := FALSE;
       #T_DataFromSafetyCard.Byte0_Bit0_QBadCh0 := FALSE;
       #T_DataFromSafetyCard.Byte0_Bit1_QBadCh1 := FALSE;
       #T_DataFromSafetyCard.Byte0_Bit2_QBadCh2 := FALSE;
       #T_DataFromSafetyCard.Byte0_Bit3_QBadCh3 := FALSE;
   END_IF;
END_REGION

REGION Network 5: **** 1 - Inputs ****Qbad Channel 0
   // Qbad Channel 0
   #QbadCh0 := (NOT #T_DataFromSafetyCard.Byte1_Bit0_QBadCh0 AND NOT #C_OutputCard) OR (NOT #T_DataFromSafetyCard.Byte0_Bit0_QBadCh0 AND #C_OutputCard);
END_REGION

REGION Network 6: **** 1 - Inputs **** Qbad Channel 1
   // Qbad Channel 1
   #QbadCh1 := (NOT #T_DataFromSafetyCard.Byte1_Bit1_QBadCh1 AND NOT #C_OutputCard) OR (NOT #T_DataFromSafetyCard.Byte0_Bit1_QBadCh1 AND #C_OutputCard);
END_REGION

REGION Network 7: **** 1 - Inputs **** Qbad Channel 2
   // Qbad Channel 2
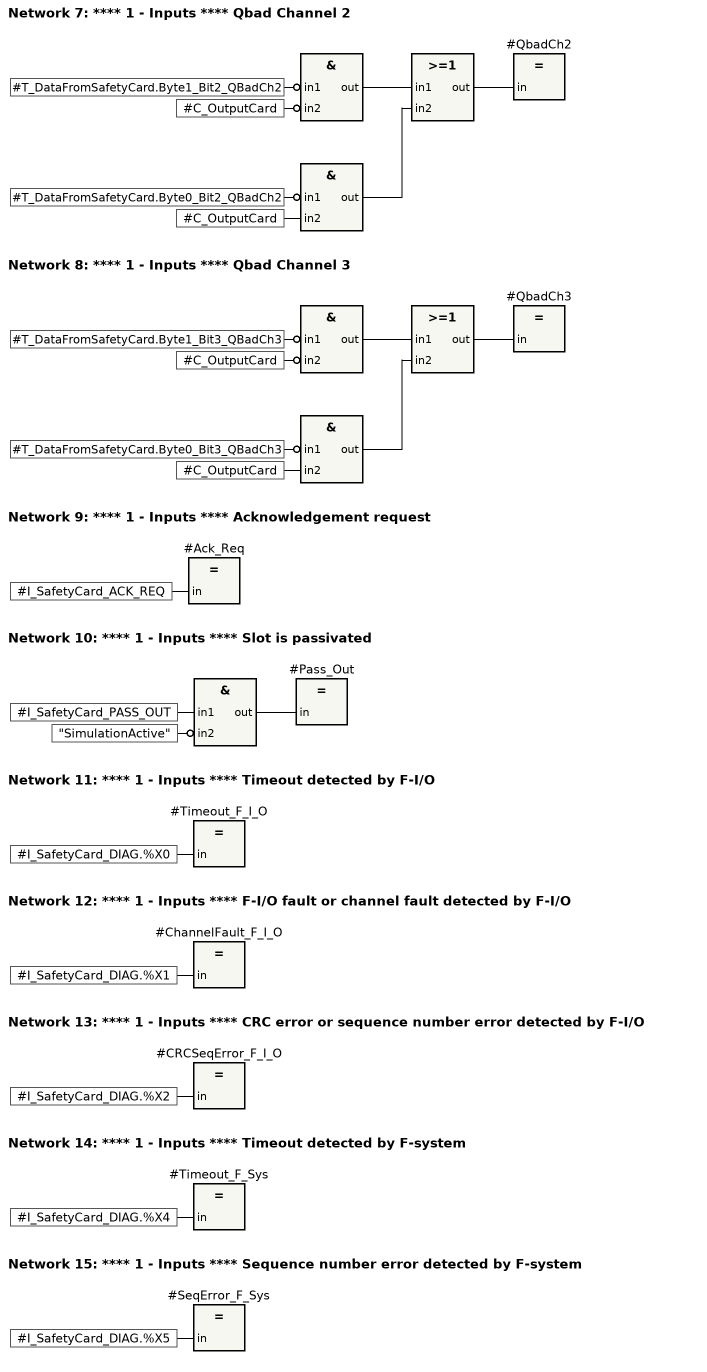
   #QbadCh2 := (NOT #T_DataFromSafetyCard.Byte1_Bit2_QBadCh2 AND NOT #C_OutputCard) OR (NOT #T_DataFromSafetyCard.Byte0_Bit2_QBadCh2 AND #C_OutputCard);
END_REGION

REGION Network 8: **** 1 - Inputs **** Qbad Channel 3
   // Qbad Channel 3
   #QbadCh3 := (NOT #T_DataFromSafetyCard.Byte1_Bit3_QBadCh3 AND NOT #C_OutputCard) OR (NOT #T_DataFromSafetyCard.Byte0_Bit3_QBadCh3 AND #C_OutputCard);
END_REGION

REGION Network 9: **** 1 - Inputs **** Acknowledgement request
   // Acknowledgement request
   #Ack_Req := #I_SafetyCard_ACK_REQ;
END_REGION

REGION Network 10: **** 1 - Inputs **** Slot is passivated
   // Slot is passivated
   #Pass_Out := #I_SafetyCard_PASS_OUT AND NOT "SimulationActive";
END_REGION

REGION Network 11: **** 1 - Inputs **** Timeout detected by F-I/O
   // Timeout detected by F-I/O
   #Timeout_F_I_O := #I_SafetyCard_DIAG.%X0;
END_REGION

REGION Network 12: **** 1 - Inputs **** F-I/O fault or channel fault detected by F-I/O
   // F-I/O fault or channel fault detected by F-I/O
   #ChannelFault_F_I_O := #I_SafetyCard_DIAG.%X1;
END_REGION

REGION Network 13: **** 1 - Inputs **** CRC error or sequence number error detected by F-I/O
   // CRC error or sequence number error detected by F-I/O
   #CRCSeqError_F_I_O := #I_SafetyCard_DIAG.%X2;
END_REGION

REGION Network 14: **** 1 - Inputs **** Timeout detected by F-system
   // Timeout detected by F-system
   #Timeout_F_Sys := #I_SafetyCard_DIAG.%X4;
END_REGION

REGION Network 15: **** 1 - Inputs **** Sequence number error detected by F-system
   // Sequence number error detected by F-system
   #SeqError_F_Sys := #I_SafetyCard_DIAG.%X5;
END_REGION

REGION Network 16: **** 1 - Inputs **** CRC error detected by F-system
   // CRC error detected by F-system
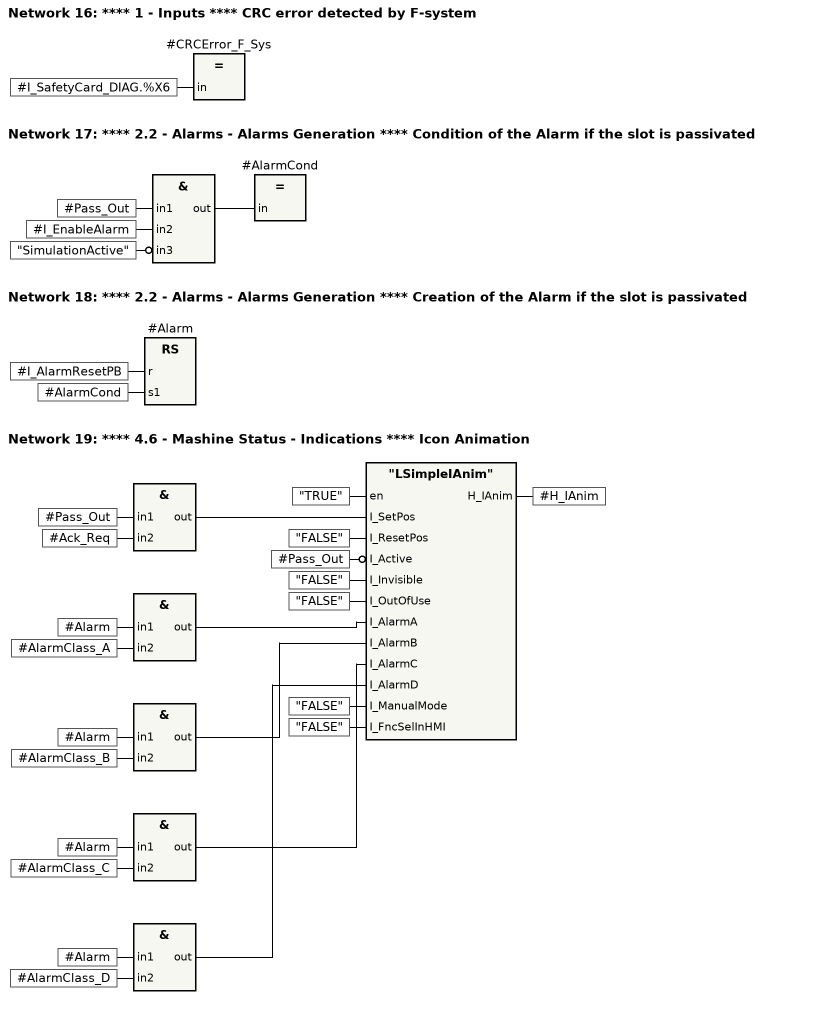
   #CRCError_F_Sys := #I_SafetyCard_DIAG.%X6;
END_REGION

REGION Network 17: **** 2.2 - Alarms - Alarms Generation **** Condition of the Alarm if the slot is passivated
   // Condition of the Alarm if the slot is passivated
   #AlarmCond := #Pass_Out AND #I_EnableAlarm AND NOT "SimulationActive";
END_REGION

REGION Network 18: **** 2.2 - Alarms - Alarms Generation **** Creation of the Alarm if the slot is passivated
   // Creation of the Alarm if the slot is passivated
   IF #I_AlarmResetPB THEN
       #Alarm := FALSE;   // RS flip-flop
   END_IF;
   IF #AlarmCond THEN #Alarm := TRUE; END_IF;
END_REGION

REGION Network 19: **** 4.6 - Mashine Status - Indications **** Icon Animation
   // Icon Animation
   IF "TRUE" THEN
       "LSimpleIAnim"(I_SetPos := #Pass_Out AND #Ack_Req,
                      I_ResetPos := "FALSE",
                      I_Active := NOT #Pass_Out,
                      I_Invisible := "FALSE",
                      I_OutOfUse := "FALSE",
                      I_AlarmA := #Alarm AND #AlarmClass_A,
                      I_AlarmB := #Alarm AND #AlarmClass_B,
                      I_AlarmC := #Alarm AND #AlarmClass_C,
                      I_AlarmD := #Alarm AND #AlarmClass_D,
                      I_ManualMode := "FALSE",
                      I_FncSelInHMI := "FALSE",
                      H_IAnim => #H_IAnim);
   END_IF;
END_REGION

REGION Network 20: **** 4.6 - Mashine Status - Indications **** Animation
   // Animation
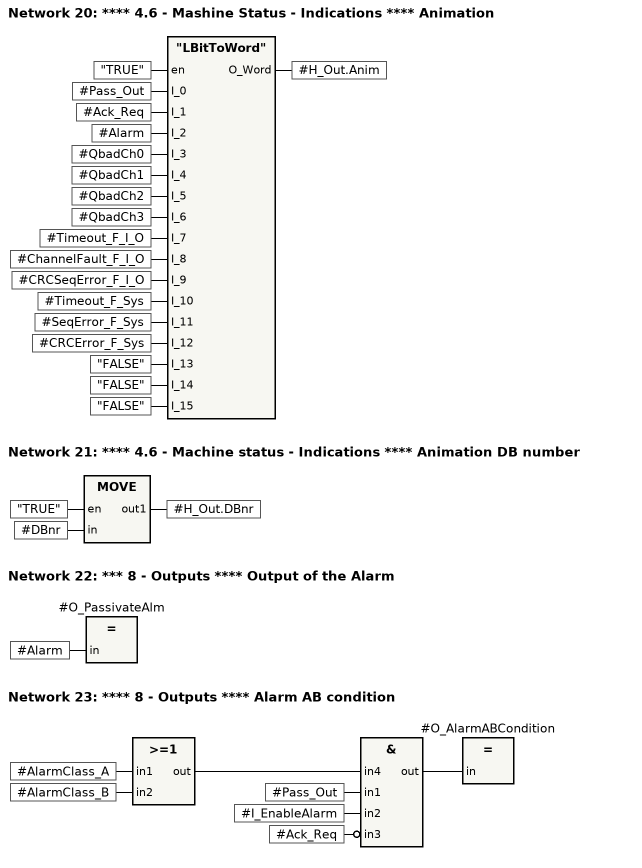
   IF "TRUE" THEN
       "LBitToWord"(I_0 := #Pass_Out,
                    I_1 := #Ack_Req,
                    I_2 := #Alarm,
                    I_3 := #QbadCh0,
                    I_4 := #QbadCh1,
                    I_5 := #QbadCh2,
                    I_6 := #QbadCh3,
                    I_7 := #Timeout_F_I_O,
                    I_8 := #ChannelFault_F_I_O,
                    I_9 := #CRCSeqError_F_I_O,
                    I_10 := #Timeout_F_Sys,
                    I_11 := #SeqError_F_Sys,
                    I_12 := #CRCError_F_Sys,
                    I_13 := "FALSE",
                    I_14 := "FALSE",
                    I_15 := "FALSE",
                    O_Word => #H_Out.Anim);
   END_IF;
END_REGION

REGION Network 21: **** 4.6 - Machine status - Indications **** Animation DB number
   // Animation DB number
   IF "TRUE" THEN #H_Out.DBnr := #DBnr; END_IF;
END_REGION

REGION Network 22: *** 8 - Outputs **** Output of the Alarm
   // Output of the Alarm
   #O_PassivateAlm := #Alarm;
END_REGION

REGION Network 23: **** 8 - Outputs **** Alarm AB condition
   // Alarm AB condition
   #O_AlarmABCondition := (#AlarmClass_A OR #AlarmClass_B) AND #Pass_Out AND #I_EnableAlarm AND NOT #Ack_Req;
END_REGION
END_FUNCTION_BLOCK

FUNCTION_BLOCK "L1SafetyCh1Alarm"   // FB1421, FBD
TITLE = L1SafetyCh1Alarm
{ S7_Optimized_Access := 'FALSE' }
AUTHOR : VCC
FAMILY : AlarmHnd
NAME : 1SafeAlm
VERSION : 0.1
// ================================================================================
// This module is used everywhere one alarm shall be generated when one security 
// input becomes False.
// The alarm can be True only when the input Enable Alarm is also True.
// When the condition to generate the alarm is not fullfilled, a boolean output is 
// available to inform the upper level that the alarm can be reset.
// The alarm is reset by means of the AlarmResetPB signal.
// 
// This module generates also a word containing all necessary information for HMI 
// Icon animation, and a word with all information for HMI safety module 
// diagnostic 
// screen. 
// ================================================================================
// stored: AutoNumber false, IsIECCheckEnabled false, SetENOAutomatically False, UDAEnableTagReadback false
   VAR_INPUT
      I_Input { ExternalAccessible := 'False'; ExternalVisible := 'False'; ExternalWritable := 'False'} : Bool;   // Input safety alarm (normally closed)
      I_AlarmClass { ExternalAccessible := 'False'; ExternalVisible := 'False'; ExternalWritable := 'False'} : Char;   // Alarm class -> A - B - C - D or E
      I_EnableAlarm { ExternalAccessible := 'False'; ExternalVisible := 'False'; ExternalWritable := 'False'} : Bool := TRUE;   // Enable alarm from upper level (0=disable/1=enable)
      I_AlarmResetPB { ExternalAccessible := 'False'; ExternalVisible := 'False'; ExternalWritable := 'False'} : Bool;   // Alarm reset pushbutton is activated
      I_SafetyCard_PASS_OUT { ExternalAccessible := 'False'; ExternalVisible := 'False'; ExternalWritable := 'False'} : Bool;   // Automatically generated DB from F-Modul (F-Peripherie DB)
      I_SafetyCard_ACK_REQ { ExternalAccessible := 'False'; ExternalVisible := 'False'; ExternalWritable := 'False'} : Bool;   // Automatically generated DB from F-Modul (F-Peripherie DB)
      I_SafetyCard_DIAG { ExternalAccessible := 'False'; ExternalVisible := 'False'; ExternalWritable := 'False'} : Byte;   // Automatically generated DB from F-Modul (F-Peripherie DB)
      I_SafetyCardHWSub { ExternalAccessible := 'False'; ExternalVisible := 'False'; ExternalWritable := 'False'} : HW_SUBMODULE;   // Safety I/O connection hardware
      I_ChannelNr { ExternalAccessible := 'False'; ExternalVisible := 'False'; ExternalWritable := 'False'} : Int;   // Used Channel Nr (Value : 0 - 7)
   END_VAR
   VAR_OUTPUT
      O_Alarm { ExternalAccessible := 'False'; ExternalVisible := 'False'; ExternalWritable := 'False'} : Bool;   // Alarm
      O_AlarmABCondition { ExternalAccessible := 'False'; ExternalVisible := 'False'; ExternalWritable := 'False'} : Bool;   // Alarm AB condition
      H_IAnim { ExternalAccessible := 'False'; ExternalVisible := 'False'; ExternalWritable := 'False'} : Word;   // Icon Animation
   END_VAR
   VAR DB_SPECIFIC
      H_Out : Struct   // HMI
         Anim : Word;   // HMI Animation of the object
         DBnr : Int;   // HMI Animation DB number
      END_STRUCT;
      Alarm { ExternalAccessible := 'False'; ExternalVisible := 'False'; ExternalWritable := 'False'} : Bool;   // Alarm
      AlarmClass_A { ExternalAccessible := 'False'; ExternalVisible := 'False'; ExternalWritable := 'False'} : Bool;   // The alarm is from alarm class A
      AlarmClass_B { ExternalAccessible := 'False'; ExternalVisible := 'False'; ExternalWritable := 'False'} : Bool;   // The alarm is from alarm class B
      AlarmClass_C { ExternalAccessible := 'False'; ExternalVisible := 'False'; ExternalWritable := 'False'} : Bool;   // The alarm is from alarm class C
      AlarmClass_D { ExternalAccessible := 'False'; ExternalVisible := 'False'; ExternalWritable := 'False'} : Bool;   // The alarm is from alarm class D
      QbadCh1 { ExternalAccessible := 'False'; ExternalVisible := 'False'; ExternalWritable := 'False'} : Bool;   // Passivation first Channel
      Ack_Req { ExternalAccessible := 'False'; ExternalVisible := 'False'; ExternalWritable := 'False'} : Bool;   // Acknowledgement request
      Timeout_F_I_O { ExternalAccessible := 'False'; ExternalVisible := 'False'; ExternalWritable := 'False'} : Bool;   // Timeout detected by F-I/O
      ChannelFault_F_I_O { ExternalAccessible := 'False'; ExternalVisible := 'False'; ExternalWritable := 'False'} : Bool;   // F-I/O fault or channel fault detected by F-I/O
      CRCSeqError_F_I_O { ExternalAccessible := 'False'; ExternalVisible := 'False'; ExternalWritable := 'False'} : Bool;   // CRC error or sequence number error detected by F-I/O
      Timeout_F_Sys { ExternalAccessible := 'False'; ExternalVisible := 'False'; ExternalWritable := 'False'} : Bool;   // Timeout detected by F-System
      SeqError_F_Sys { ExternalAccessible := 'False'; ExternalVisible := 'False'; ExternalWritable := 'False'} : Bool;   // Sequence number error detected by F-system
      CRCError_F_Sys { ExternalAccessible := 'False'; ExternalVisible := 'False'; ExternalWritable := 'False'} : Bool;   // CRC error detected by F-system
      AlarmCond { ExternalAccessible := 'False'; ExternalVisible := 'False'; ExternalWritable := 'False'} : Bool;   // Alarm condition
      RetValueData { ExternalAccessible := 'False'; ExternalVisible := 'False'; ExternalWritable := 'False'} : Int;   // Status variable (SFC14)
      DBnr { ExternalAccessible := 'False'; ExternalVisible := 'False'; ExternalWritable := 'False'} : Int;   // HMI DB number
   END_VAR
   VAR_TEMP
      T_DataFromSafetyCard : Struct   // Temp structure : receive data's from Safety Card
         Byte0_Bit0_Spare : Bool;
         Byte0_Bit1_Spare : Bool;
         Byte0_Bit2_Spare : Bool;
         Byte0_Bit3_Spare : Bool;
         Byte0_Bit4_Spare : Bool;
         Byte0_Bit5_Spare : Bool;
         Byte0_Bit6_Spare : Bool;
         Byte0_Bit7_Spare : Bool;
         Byte1_Bit0_QBadCh0 : Bool;
         Byte1_Bit1_QBadCh1 : Bool;
         Byte1_Bit2_QBadCh2 : Bool;
         Byte1_Bit3_QBadCh3 : Bool;
         Byte1_Bit4_QBadCh4 : Bool;
         Byte1_Bit5_QBadCh5 : Bool;
         Byte1_Bit6_QBadCh6 : Bool;
         Byte1_Bit7_QBadCh7 : Bool;
         Byte2_bit0_Spare : Bool;
         Byte2_bit1_Spare : Bool;
         Byte2_bit2_Spare : Bool;
         Byte2_bit3_Spare : Bool;
         Byte2_bit4_Spare : Bool;
         Byte2_bit5_Spare : Bool;
         Byte2_bit6_Spare : Bool;
         Byte2_bit7_Spare : Bool;
         Byte3_Bit0_Spare : Bool;
         Byte3_Bit1_Spare : Bool;
         Byte3_Bit2_Spare : Bool;
         Byte3_Bit3_Spare : Bool;
         Byte3_Bit4_Spare : Bool;
         Byte3_Bit5_Spare : Bool;
         Byte3_Bit6_Spare : Bool;
         Byte3_Bit7_Spare : Bool;
         Byte4_bit0_Spare : Bool;
         Byte4_bit1_Spare : Bool;
         Byte4_bit2_Spare : Bool;
         Byte4_bit3_Spare : Bool;
         Byte4_bit4_Spare : Bool;
         Byte4_bit5_Spare : Bool;
         Byte4_bit6_Spare : Bool;
         Byte4_bit7_Spare : Bool;
         Byte5_bit0_Spare : Bool;
         Byte5_bit1_Spare : Bool;
         Byte5_bit2_Spare : Bool;
         Byte5_bit3_Spare : Bool;
         Byte5_bit4_Spare : Bool;
         Byte5_bit5_Spare : Bool;
         Byte5_bit6_Spare : Bool;
         Byte5_bit7_Spare : Bool;
      END_STRUCT;
   END_VAR
BEGIN

NETWORK
TITLE = **** 1 - Inputs **** DB number
// DB number
      L     DINO;
      T     #DBnr;

NETWORK
TITLE = **** 1 - Inputs **** Alarm class
// Alarm class
// Alarm class = D
      L     #I_AlarmClass;
      L     'D';
      ==I;
      =     #AlarmClass_D;

// Alarm class = C
      L     #I_AlarmClass;
      L     'C';
      ==I;
      =     #AlarmClass_C;

// Alarm class = B
      L     #I_AlarmClass;
      L     'B';
      ==I;
      =     #AlarmClass_B;

// Alarm class = A
      AN    #AlarmClass_B;
      AN    #AlarmClass_C;
      AN    #AlarmClass_D;
      =     #AlarmClass_A;


REGION Network 3: **** 1 - Inputs **** Safety I/O connection hardware
   // Safety I/O connection hardware
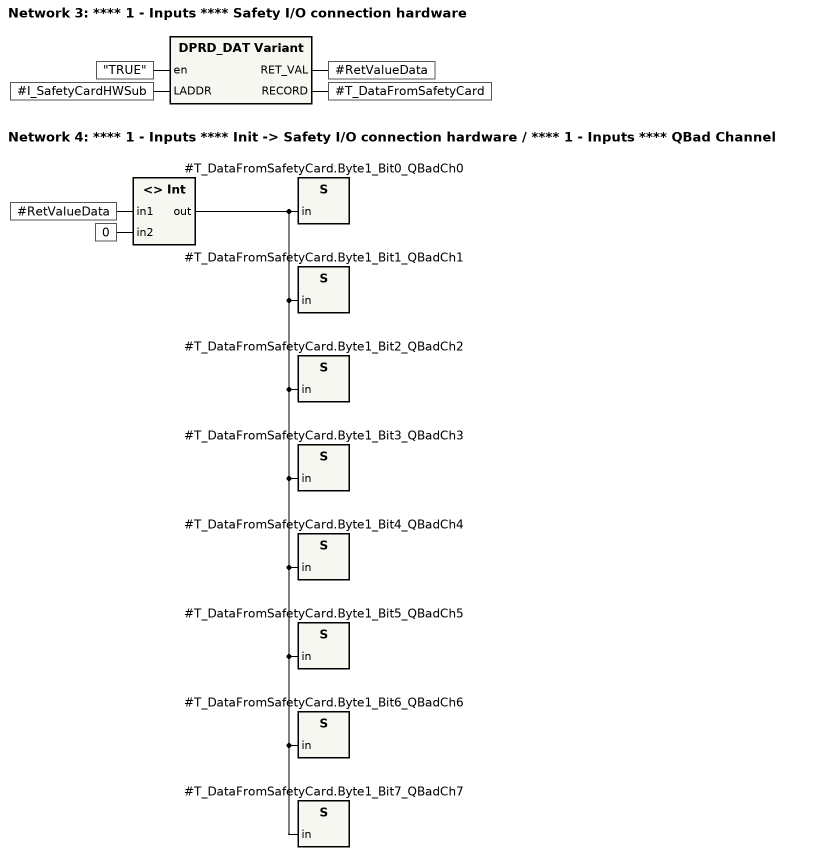
   IF "TRUE" THEN
       #RetValueData := DPRD_DAT(LADDR := #I_SafetyCardHWSub, RECORD => #T_DataFromSafetyCard);
   END_IF;
END_REGION

REGION Network 4: **** 1 - Inputs **** Init -> Safety I/O connection hardware / **** 1 - Inputs **** QBad Channel
   // Init -> Safety I/O connection hardware
   IF #RetValueData <> 0 THEN
       #T_DataFromSafetyCard.Byte1_Bit0_QBadCh0 := TRUE;
       #T_DataFromSafetyCard.Byte1_Bit1_QBadCh1 := TRUE;
       #T_DataFromSafetyCard.Byte1_Bit2_QBadCh2 := TRUE;
       #T_DataFromSafetyCard.Byte1_Bit3_QBadCh3 := TRUE;
       #T_DataFromSafetyCard.Byte1_Bit4_QBadCh4 := TRUE;
       #T_DataFromSafetyCard.Byte1_Bit5_QBadCh5 := TRUE;
       #T_DataFromSafetyCard.Byte1_Bit6_QBadCh6 := TRUE;
       #T_DataFromSafetyCard.Byte1_Bit7_QBadCh7 := TRUE;
   END_IF;
END_REGION

REGION Network 5: **** 1 - Inputs **** Qbad Channel 1
   // Qbad Channel 1
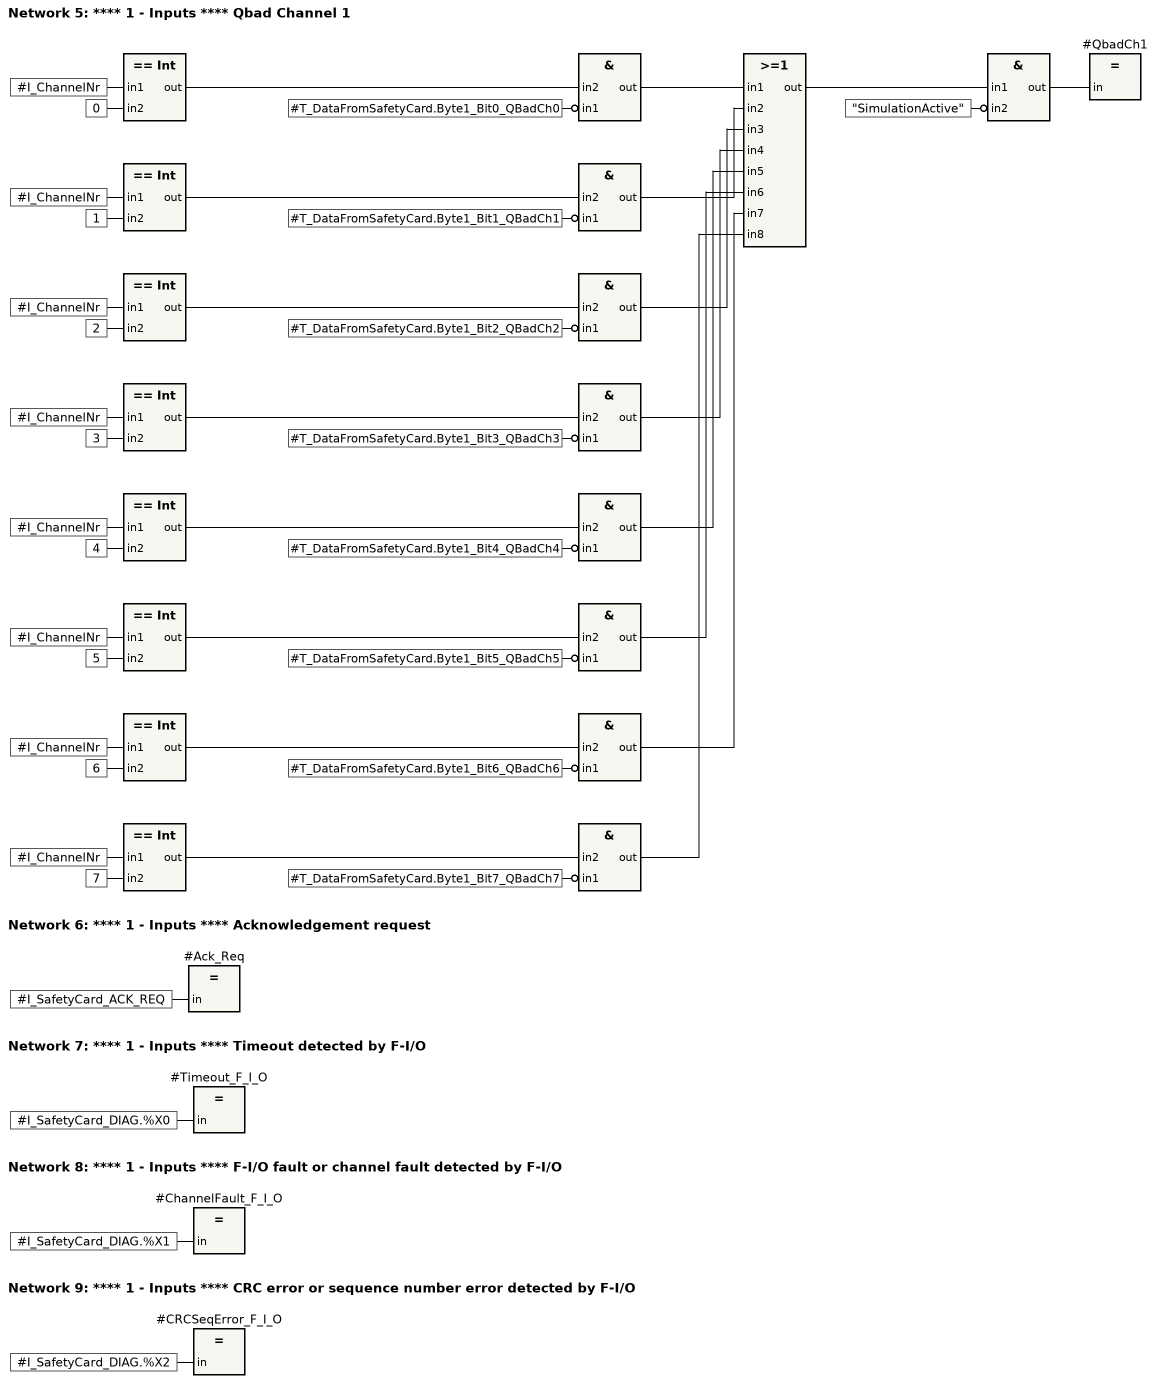
   #QbadCh1 := (((#I_ChannelNr = 0) AND NOT #T_DataFromSafetyCard.Byte1_Bit0_QBadCh0) OR ((#I_ChannelNr = 1) AND NOT #T_DataFromSafetyCard.Byte1_Bit1_QBadCh1) OR ((#I_ChannelNr = 2) AND NOT #T_DataFromSafetyCard.Byte1_Bit2_QBadCh2) OR ((#I_ChannelNr = 3) AND NOT #T_DataFromSafetyCard.Byte1_Bit3_QBadCh3) OR ((#I_ChannelNr = 4) AND NOT #T_DataFromSafetyCard.Byte1_Bit4_QBadCh4) OR ((#I_ChannelNr = 5) AND NOT #T_DataFromSafetyCard.Byte1_Bit5_QBadCh5) OR ((#I_ChannelNr = 6) AND NOT #T_DataFromSafetyCard.Byte1_Bit6_QBadCh6) OR ((#I_ChannelNr = 7) AND NOT #T_DataFromSafetyCard.Byte1_Bit7_QBadCh7)) AND NOT "SimulationActive";
END_REGION

REGION Network 6: **** 1 - Inputs **** Acknowledgement request
   // Acknowledgement request
   #Ack_Req := #I_SafetyCard_ACK_REQ;
END_REGION

REGION Network 7: **** 1 - Inputs **** Timeout detected by F-I/O
   // Timeout detected by F-I/O
   #Timeout_F_I_O := #I_SafetyCard_DIAG.%X0;
END_REGION

REGION Network 8: **** 1 - Inputs **** F-I/O fault or channel fault detected by F-I/O
   // F-I/O fault or channel fault detected by F-I/O
   #ChannelFault_F_I_O := #I_SafetyCard_DIAG.%X1;
END_REGION

REGION Network 9: **** 1 - Inputs **** CRC error or sequence number error detected by F-I/O
   // CRC error or sequence number error detected by F-I/O
   #CRCSeqError_F_I_O := #I_SafetyCard_DIAG.%X2;
END_REGION

REGION Network 10: **** 1 - Inputs **** Timeout detected by F-system
   // Timeout detected by F-system
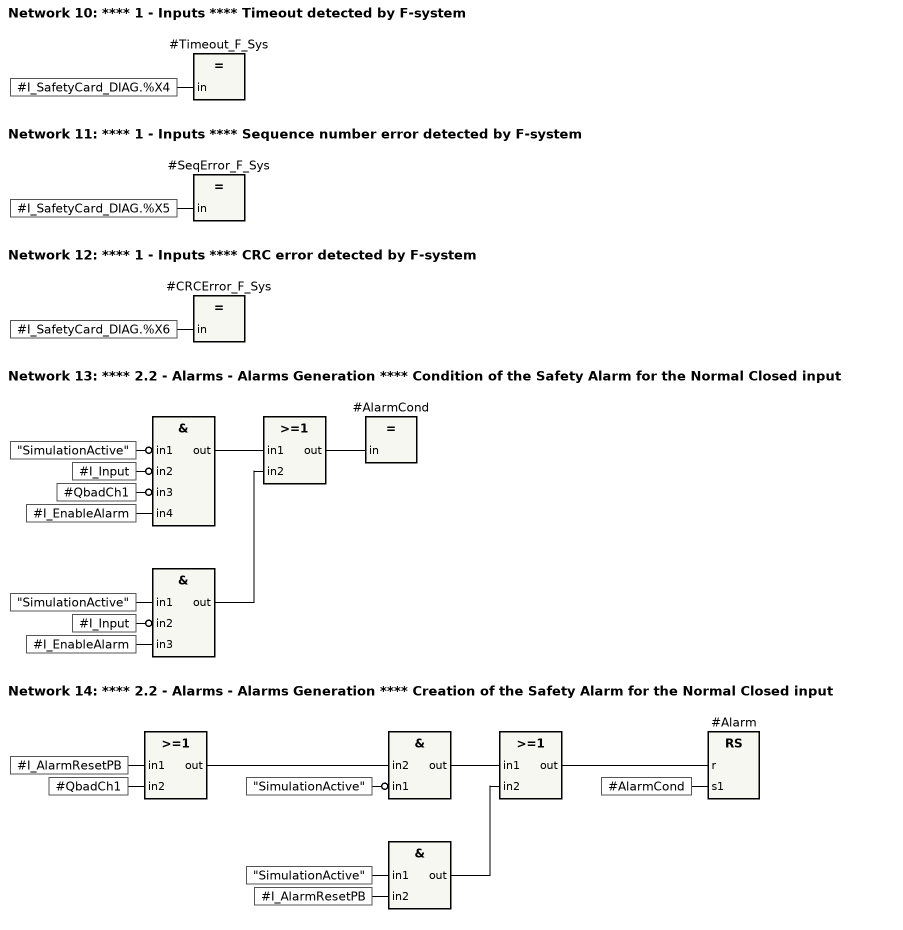
   #Timeout_F_Sys := #I_SafetyCard_DIAG.%X4;
END_REGION

REGION Network 11: **** 1 - Inputs **** Sequence number error detected by F-system
   // Sequence number error detected by F-system
   #SeqError_F_Sys := #I_SafetyCard_DIAG.%X5;
END_REGION

REGION Network 12: **** 1 - Inputs **** CRC error detected by F-system
   // CRC error detected by F-system
   #CRCError_F_Sys := #I_SafetyCard_DIAG.%X6;
END_REGION

REGION Network 13: **** 2.2 - Alarms - Alarms Generation **** Condition of the Safety Alarm for the Normal Closed input
   // Condition of the Safety Alarm for the Normal Closed input
   #AlarmCond := (NOT "SimulationActive" AND NOT #I_Input AND NOT #QbadCh1 AND #I_EnableAlarm) OR ("SimulationActive" AND NOT #I_Input AND #I_EnableAlarm);
END_REGION

REGION Network 14: **** 2.2 - Alarms - Alarms Generation **** Creation of the Safety Alarm for the Normal Closed input
   // Creation of the Safety Alarm for the Normal Closed input
   IF ((#I_AlarmResetPB OR #QbadCh1) AND NOT "SimulationActive") OR ("SimulationActive" AND #I_AlarmResetPB) THEN
       #Alarm := FALSE;   // RS flip-flop
   END_IF;
   IF #AlarmCond THEN #Alarm := TRUE; END_IF;
END_REGION

REGION Network 15: **** 4.6 - Mashine Status - Indications **** Icon Animation
   // Icon Animation
